# B&R Automation Studio project PrintMarkCC_LW3
Automation Studio 4.12.4.107 SP; technology packages: Acp10Arnc0 5.23.1, mapp 5.23.1, mappView 5.23.0

## Configuration Config1

### Task classes (Cpu.sw)
```
Cyclic#4:
  Cutter <- Cutter.Cutter.prg
  ConvCtrl <- ConvCtrl.ConvCtrl.prg
  AlarmsX <- Alarms.AlarmsX.prg
DataObjects: Acp10sys
NcDataObjects: gAxMsa <- Axis.gAxMaster.gAxMsa.dob, gAxMsi <- Axis.gAxMaster.gAxMsi.dob, acp10etxen <- Axis.acp10etxen.dob, gAxSlavea <- Axis.gAxSlave.gAxSlavea.dob, gAxSlavei <- Axis.gAxSlave.gAxSlavei.dob
Binaries: arsvcreg, udbdef, TCData, FWRules, Acp10map, acp10cfg, ashwd, slaveaxis, ashwac, User, sysconf, asfw, arconfig, masteraxis, iomap, Role
Libraries: Acp10man, Acp10par, NcGlobal, MpAxis, Acp10_MC, MpBase, MpCom, sys_lib, brsystem, runtime, MC_RegMa, MpAlarmX, astime, asieccon, powerlnk, asbrstr, fileio, dataobj
```

### masteraxis.mpaxisbasic - X20CP0484/Motion/masteraxis.mpaxisbasic
```
Element gmlMaster (Type=mpaxisbasic)
```

### slaveaxis.mpaxisbasic - X20CP0484/Motion/slaveaxis.mpaxisbasic
```
Element gAxisSlave (Type=mpaxisbasic)
```

## Configuration Config2

### Task classes (Cpu.sw)
```
Cyclic#1:
  Cutter <- Cutter.Cutter.prg  // cutter axis control
  ConvCtrl <- ConvCtrl.ConvCtrl.prg  // conveyor control
  AutoCtrl <- AutoCtrl.AutoCtrl.prg  // main control
Cyclic#8:
  AlarmsX <- Alarms.AlarmsX.prg  // alarm funcitons
  DataRec <- Datarec.DataRec.prg  // data recorder
DataObjects: Acp10sys
NcDataObjects: gAxMsa <- Axis.gAxMaster.gAxMsa.dob, gAxMsi <- Axis.gAxMaster.gAxMsi.dob, acp10etxen <- Axis.acp10etxen.dob, gAxSlavea <- Axis.gAxSlave.gAxSlavea.dob, gAxSlavei <- Axis.gAxSlave.gAxSlavei.dob
Binaries: arsvcreg, udbdef, TCData, FWRules, mvLoader, arflatprv, TCLang, arcoal, Acp10map, acp10cfg, ashwd, slaveaxis, ashwac, User, sysconf, asfw, arconfig, masteraxis, iomap, Role, Alarms, UserX, TC, dataReco
Libraries: Acp10man, Acp10par, NcGlobal, MpAxis, Acp10_MC, MpBase, MpCom, sys_lib, brsystem, runtime, MC_RegMa, MpAlarmX, astime, MpUserX, MpData, FileIO, DataObj, asieccon, powerlnk, asbrstr, arcert, aseth, ashw, aruser, arssl
```

### slaveaxis.mpaxisbasic - X20CP0484/Motion/slaveaxis.mpaxisbasic
```
Element gmlSlave (Type=mpaxisbasic)
```

### Alarms.mpalarmxcore - X20CP0484/mappServices/Alarms.mpalarmxcore
```
Element gAlarmXCore (Type=mpalarmxcore)
  mapp.AlarmX.Core.Configuration:
    [0]:
      Name = InTheCuttingZone
      Message = axis is inside the cutting zone please move it manually
      Code = 55
      Severity = 100
      Behavior = PersistentAlarm
    [1]:
      Name = ErrorCutting
      Code = 65
      Severity = 100
      Behavior = PersistentAlarm
```

### UserX.mpuserx - X20CP0484/mappServices/UserX.mpuserx
```
Element UserMgmtX (Type=mpuserx)
  ServerSettings:
    Server:
      AdditionalUserData:
        [0] = mail
        [1] = telephoneNumber
  Users:
    DefUser#1:
      id = admin
      name = admin
      lang = en
  Groups:
    DefGroup#1:
      id = Administrators
      level = 100
      admin = TRUE
      rights:
        [0] = FullAccess
    DefGroup#2:
      id = Everyone
    DefGroup#3:
      id = Operator
      level = 80
      rights:
        [0] = FullAccess
    DefGroup#4:
      id = Service
      level = 50
      rights:
        [0] = FullAccess
```

## Configuration Config3

### Task classes (Cpu.sw)
```
Cyclic#1:
  Cutter <- Cutter.Cutter.prg  // cutter axis control
  ConvCtrl <- ConvCtrl.ConvCtrl.prg  // conveyor control
  AutoCtrl <- AutoCtrl.AutoCtrl.prg  // main control
Cyclic#8:
  AlarmsX <- Alarms.AlarmsX.prg  // alarm funcitons
  DataRec <- Datarec.DataRec.prg  // data recorder
DataObjects: Acp10sys
NcDataObjects: gAxMsa <- Axis.gAxMaster.gAxMsa.dob, gAxMsi <- Axis.gAxMaster.gAxMsi.dob, acp10etxen <- Axis.acp10etxen.dob, gAxSlavea <- Axis.gAxSlave.gAxSlavea.dob, gAxSlavei <- Axis.gAxSlave.gAxSlavei.dob
Binaries: arsvcreg, udbdef, TCData, FWRules, mvLoader, arflatprv, TCLang, arcoal, Acp10map, acp10cfg, ashwd, slaveaxis, ashwac, User, sysconf, asfw, arconfig, masteraxis, iomap, Role, Alarms, UserX, TC, dataReco
Libraries: Acp10man, Acp10par, NcGlobal, MpAxis, Acp10_MC, MpBase, MpCom, sys_lib, brsystem, runtime, MC_RegMa, MpAlarmX, astime, MpUserX, MpData, FileIO, DataObj, asieccon, powerlnk, arcert, aseth, ashw, aruser, arssl, AsBrStr, MpServer, MpPackML
```

### Acp10map.ncm - X20CP0484/Motion/Acp10map.ncm
```
NcMapping (NcSwId=Acp10, DisabledNodesAreHidden=False)
  NcObject gAxSlave (ModuleId=8V1010.00-2a, Type=ncAXIS, Channel=1, AcoposSimulation=Off, InitParameter=gAxSlavei, AcoposParameter=gAxSlavea, AdditionalData=PLCopen_ModPos="3600,1" , Disabled=FALSE, ModuleDisabled=FALSE)
  NcObject 8V1010.00-2a_ncV_AXIS1 (ModuleId=8V1010.00-2a, Type=ncV_AXIS, Channel=1, Disabled=TRUE, ModuleDisabled=FALSE)
  NcObject gAxMaster (ModuleId=8V1010.00-2, Type=ncAXIS, Channel=1, AcoposSimulation=Off, InitParameter=gAxMsi, AcoposParameter=gAxMsa, Disabled=FALSE, ModuleDisabled=FALSE)
  NcObject 8V1010.00-2_ncV_AXIS1 (ModuleId=8V1010.00-2, Type=ncV_AXIS, Channel=1, Disabled=TRUE, ModuleDisabled=FALSE)
```

### slaveaxis.mpaxisbasic - X20CP0484/Motion/slaveaxis.mpaxisbasic
```
Element gmlSlave (Type=mpaxisbasic)
  Alarms = MpAlarmX
```

### UserX.mpuserx - X20CP0484/mappServices/UserX.mpuserx
```
Element UserMgmtX (Type=mpuserx)
  ServerSettings:
    Server:
      AdditionalUserData:
        [0] = mail
        [1] = telephoneNumber
  Users:
    DefUser#1:
      id = admin
      name = admin
      lang = en
    DefUser#2:
      id = operator
      name = operator
      lang = en
  Groups:
    DefGroup#1:
      id = Administrators
      level = 100
      admin = TRUE
      rights:
        [0] = FullAccess
    DefGroup#2:
      id = Everyone
    DefGroup#3:
      id = Operator
      level = 80
      rights:
        [0] = FullAccess
    DefGroup#4:
      id = Service
      level = 50
      rights:
        [0] = FullAccess
```

### mlPack.mppackmlcore - X20CP0484/mappServices/mlPack.mppackmlcore
```
Element gPackMLCore (Type=mppackmlcore)
  Modes:
    Mode[1]:
      ModeID = 1
      Name = Production
```

## Logical view

Binary libraries used (declarations not repeated): operator, runtime, astime, AsIecCon, Acp10man, Acp10par, NcGlobal, MpAxis, Acp10_MC, MpBase, MpCom, sys_lib, brsystem, MC_RegMa, MpAlarmX, MpUserX, MpData, FileIO, DataObj

### Global.typ - Global data types
```iecst
(*main control*)

TYPE
	AxisCtrl_typ : 	STRUCT  (*Axis Ctrl Struture*)
		Cmd : AxisCmd_typ; (*Axis Ctrl CMd type*)
		Para : AxisPara_typ; (*Axis para type*)
		Status : AxisStatus_typ; (*Axis Status Type*)
	END_STRUCT;
END_TYPE

(*commands*)

TYPE
	AxisCmd_typ : 	STRUCT  (*Axis Ctrl CMd type*)
		Start : BOOL; (*Start Cmd*)
		Stop : BOOL; (*Stop cmd*)
		PrintMark : BOOL; (*Print mark detection bit*)
		ErrorReset : BOOL; (*Error reset*)
		AutoMode : BOOL; (*AutoMode*)
		JogFwd : BOOL; (*Jog forward command*)
		JogBack : BOOL; (*jog BAckward c0mmand*)
		Home : BOOL; (*home Cmd*)
		SingleCutter : BOOL;
	END_STRUCT;
END_TYPE

(*parameters*)

TYPE
	AxisPara_typ : 	STRUCT  (*Axis para type*)
		Speed : UINT; (*Axis Speed*)
	END_STRUCT;
END_TYPE

(*status*)

TYPE
	AxisStatus_typ : 	STRUCT  (*Axis Status*)
		JogNegReady : BOOL; (*Axis jog neg ready status*)
		JogPosReady : BOOL; (*axis jog pos ready Statsus*)
	END_STRUCT;
END_TYPE
```

### Global.var - Global variables
```iecst
(*Axis Variables*)
VAR
	gAxMaster : ACP10AXIS_typ; (*Master Axis*)
	gAxSlave : ACP10AXIS_typ; (*Slave Axis*) (*	gAx_Slave : AxisBasic_type; (*Slave Axis Structure*) (*gAx_Master : AxisBasic_type; MAster axis Structure*)
END_VAR
(*Automatic mode*)
VAR
	gAutoMode : BOOL; (*automatic mode for machine*)
	gManulMode : BOOL; (*manual mode for machine*)
END_VAR
(*IR trigger for conveyor belt*)
VAR
	gIR_Trigger : BOOL; (*trigger of IR for Conveyor axis master*)
END_VAR
(*for mappview commands given'*)
VAR
	gMi_ModeConfirm : BOOL; (*mode confirmation for hmi*)
	gMI_MODE : BOOL;
END_VAR
```


### Package Logical/Axis - Axis Package


- Data object Logical/Axis/gAxMaster/gAxMsa (Apt) - Conv Axis SPT (no source held here)

- Data object Logical/Axis/gAxMaster/gAxMsi (Ax) - COnv Axis Parameter Table (no source held here)

### Package Logical/Axis/gAxSlave - Cutter Axis Package

### Data object Logical/Axis/gAxSlave/gAxSlavei (Ax) - Cutter Axis Paramter table

#### gAxisSlave.ax
```
InitParameter (Version=5.23.1, NcSwId=ACP10)
  ACP10AXIS_typ:
    dig_in:
      level:
        reference = ncACTIV_HI
        pos_hw_end = ncACTIV_HI
        neg_hw_end = ncACTIV_HI
        trigger1 = ncACTIV_HI
        trigger2 = ncACTIV_HI
    encoder_if:
      parameter:
        count_dir = ncSTANDARD
        scaling:
          load:
            units = 3600
            rev_motor = 1
    limit:
      parameter:
        v_pos = 108000.0
        v_neg = 108000.0
        a1_pos = 1080000.0
        a2_pos = 1080000.0
        a1_neg = 1080000.0
        a2_neg = 1080000.0
        t_jolt = 0.18
        t_in_pos = 0.0
        pos_sw_end = 8388607
        neg_sw_end = -8388608
        ds_warning = 180.0
        ds_stop = 360.0
        a_stop = 1.0E+30
        dv_stop = 0.0
        dv_stop_mode = ncOFF
    controller:
      mode = ncPOSITION + ncFF
      position:
        kv = 295.0
        tn = 0.0
        t_predict = 0.0004
        t_total = 0.0004
        p_max = 1.0E+30
        i_max = 0.0
      speed:
        kv = 0.6
        tn = 0.0
        t_filter = 0.0
        isq_filter1:
          type = ncOFF
          a0 = 0.0
          a1 = 0.0
          b0 = 0.0
          b1 = 0.0
          b2 = 0.0
          c0_par_id = 0
          c1_par_id = 0
        isq_filter2:
          type = ncOFF
          a0 = 0.0
          a1 = 0.0
          b0 = 0.0
          b1 = 0.0
          b2 = 0.0
          c0_par_id = 0
          c1_par_id = 0
        isq_filter3:
          type = ncOFF
          a0 = 0.0
          a1 = 0.0
          b0 = 0.0
          b1 = 0.0
          b2 = 0.0
          c0_par_id = 0
          c1_par_id = 0
      uf:
        type = ncLINEAR + ncCORRECTION
        auto_config = ncMOTOR_PAR
        u0 = 0.0
        un = 0.0
        fn = 50.0
        k_f_slip = 0.0
      ff:
        mode = ncSTANDARD
        torque_load = 0.0
        torque_pos = 0.00623549
        torque_neg = 0.00399368
        kv_torque = 0.0016169
        inertia = 9.44476E-05
        t_filter_a = 0.0
      fb:
        mode = ncSTANDARD
        speed_mix_ratio = 0.0
        speed_kv = 0.0
      model:
        mass1:
          inertia = 0.0
          viscous_friction = 0.0
        mass2:
          inertia = 0.0
          viscous_friction = 0.0
          stiffness = 0.0
          damping = 0.0
    move:
      stop:
        parameter[0]:
          decel_ramp = ncA_LIMIT
          controller = ncON
        parameter[1]:
          decel_ramp = ncA_LIMIT
          controller = ncON
        parameter[2]:
          decel_ramp = ncA_LIMIT
          controller = ncON
        parameter[3]:
          decel_ramp = ncA_LIMIT
          controller = ncON
        quickstop:
          decel_ramp = ncA_LIMIT
          t_jolt = 0.0
        drive_error:
          decel_ramp = ncA_LIMIT
      homing:
        parameter:
          s = 0
          v_switch = 5000.0
          v_trigger = 500.0
          a = 50000.0
          mode = ncDIRECT
          edge_sw = ncPOSITIVE
          start_dir = ncPOSITIVE
          trigg_dir = ncPOSITIVE
          ref_pulse = ncOFF
          fix_dir = ncOFF
          tr_s_block = 0.0
          torque_lim = 0.0
          ds_block = 0.0
          ds_stop = 0.0
      basis:
        parameter:
          v_pos = 500.0
          v_neg = 5000.0
          a1_pos = 50000.0
          a2_pos = 50000.0
          a1_neg = 50000.0
          a2_neg = 50000.0
    message:
      text:
        parameter:
          format = ncBREAK + ncZERO
          columns = 80
          data_modul = acp10etxen
```

### Program Logical/Cutter/Cutter (IEC)

#### Main.st - Init, cyclic, exit code
```iecst
(*|ŻŻŻŻŻŻŻŻŻŻŻŻŻŻŻŻŻŻŻŻŻŻŻŻŻŻŻŻŻŻŻŻŻŻŻŻŻŻŻŻŻŻŻŻŻŻŻŻŻŻŻŻŻŻŻŻŻŻŻŻŻŻŻŻŻŻŻŻŻŻŻŻŻŻŻŻŻŻŻŻŻŻŻŻŻŻŻŻŻŻŻŻŻŻŻŻŻŻŻŻŻŻŻŻŻŻŻŻŻŻ|*)
(*| Copyright      :-  B&R Industrial Automation GmbH															 |*)
(*| Contact Person :-  maskeu																					 |*)
(*|——————————————————————————————————————————————————————————————————————————————————————————————————————————————|*)
(*| System       :-  cutter control                                                                    	 		 |*)
(*| Task Name    :-  cutter control																		  		 |*)
(*| Auther Name  :-  maskeu																						 |*)
(*| Created Date :-  December 19, 2023 																		   	 |*)
(*| Task Class   :-  Task Class# 1                                                                 				 |*)
(*| Task Time    :-  Task Timing 2mSec                                                                           |*)
(*| OS Version   :-  G4.93                                                                                       |*)
(*| AS Version   :-  AS 4.12.4.107 SP                                                                            |*)
(*|——————————————————————————————————————————————————————————————————————————————————————————————————————————————|*)
(*| Description  :-  CUTTER cam sequnce and basic initial prameters		    									 |*)
(*| V1.00.0   19/12/2023	 Maskeu        added cam sequnce 									Complete		 |*)
(*| V2.00.0   21/12/2023	 Maskeu        added basic parameters for axis						Complete		 |*)
(*| V3.00.0   22/12/2023	 Maskeu        added reg capture parameters 						Complete		 |*)
PROGRAM _INIT

	//providing initial parameters
	iBasicParSlave.Acceleration:=10800;
	iBasicParSlave.Deceleration:=108000;
	iBasicParSlave.Jog.Deceleration:=108000;
	iBasicParSlave.Jog.Acceleration:=108000;
	iBasicParSlave.Jog.Velocity:=360;

	//assigning reg capture prameters
	iRegCapAdvPar.EventSourceParID := ACP10PAR_STAT_TRIGGER1;
	iRegCapAdvPar.Edge := ncP_EDGE;
	iRegCapAdvPar.MinWidth := 50;
	iRegCapAdvPar.MaxWidth := 200;
	iRegCapAdvPar.WindowNeg := 200;
	iRegCapAdvPar.WindowPos := 200;
	iRegCapAdvPar.SensorDelay := 200;
	iRegCapAdvPar.CorrectCurrentCycle := TRUE;
	iRegCapAdvPar.CorrectionValueLimitNeg := 70;
	iRegCapAdvPar.CorrectionValueLimitPos := 70;

	iRegCapConfig.DistanceToSensor := 1050; //distance betwwen ir sensor to cutter
	iRegCapConfig.ProductLength := 700;		//length of the product
	iRegCapConfig.RegMarkPosition := 700;	//reg par at positon 7c,
	iRegCapConfig.RegMarkOffset := 10;		//offset value
END_PROGRAM

PROGRAM _CYCLIC
	IF iCutCtrl.Cmd.SingleCutter THEN
		//axis control  in single mode
		SingleCutter;
		// cam for single cutter
		CamSingle;
	ELSE
		//axis control  in dual mode
		MultCutter;
		// cam for Dual Cutter
		CamMulti;
	END_IF

	IF iFb_SlaveAx.Info.PLCopenState = mpAXIS_SYNCHRONIZED_MOTION THEN
		iFb_RegCap();
	END_IF

	//reg capturing action
	RegCap;

	//linking the slave to cam sequence
	iFb_CamSequ.MpLink :=ADR(gmlSlave);
	iFb_CamSequ.Enable :=TRUE;

	//parameters for cam seqeunce
	iFb_CamSequ.Parameters :=ADR(iAx_CamSequence);

	//linking the master with cam sequence
	iFb_CamSequ.MpLinkMaster :=ADR(gmlMaster);
	iFb_CamSequ.StartSequence :=iFb_CamSequ.Info.MasterReady AND iFb_CamSequ.Info.SlaveReady;

	//fucniton block is callled
	iFb_CamSequ();

	IF (iMI_CutSetJogAcc <> (iBasicParSlave.Jog.Acceleration * PER_SEC)/PRODUCT_LENGTH
		OR iMI_CutSetJogDeacc <> (iBasicParSlave.Jog.Deceleration  * PER_SEC)/PRODUCT_LENGTH
		OR iMI_CutSetJogVel <> (iBasicParSlave.Jog.Velocity * PER_SEC)/PRODUCT_LENGTH)
		AND NOT gMI_MODE THEN
		iFb_SlaveAx.Update := TRUE;
		IF iFb_SlaveAx.UpdateDone THEN
			iFb_SlaveAx.Update := FALSE;
		END_IF
	END_IF

	iBasicParSlave.Jog.Acceleration := (iMI_CutSetJogAcc * PRODUCT_LENGTH)/PER_SEC;
	iBasicParSlave.Jog.Deceleration := (iMI_CutSetJogDeacc * PRODUCT_LENGTH)/PER_SEC;
	iBasicParSlave.Jog.Velocity := (iMI_CutSetJogVel * PRODUCT_LENGTH)/PER_SEC;

	iMI_CutActSpeed := (iFb_SlaveAx.Velocity * PER_SEC)/PRODUCT_LENGTH ;
END_PROGRAM

PROGRAM _EXIT

	//disabling all the functions
	iFb_AxisSlave.Enable:=FALSE;
	iFb_AxisSlave();
	iFb_CamSequ.Enable:=FALSE;
	iFb_CamSequ();
END_PROGRAM
```

#### Types.typ - Local data types
```iecst
(*jog limiting enumeration*)

TYPE
	Joglim_enum :
		( (*jog limit state enumeration*)
		enCHECKVEL, (*Checking value*)
		enADDVEL, (*gicing jog values*)
		enUPPERPOS, (*upper position state*)
		enLOWERPOS, (*lower position state*)
		enUPDATE, (*updating the state according position*)
		enRESET (*reseting the values*)
		);
END_TYPE

(*axis steps enumeration*)

TYPE
	AxStep_enum :
		( (*axis enumeration*)
		enINITA, (*initiate*)
		enSTARTA, (*starting axis*)
		enNEEGHOMEMOVE, (*negative direction homing*)
		enPOWER_ONA, (*powering on*)
		enPOSHOMINGSEC, (*positive direction homing*)
		enPOSHOMING, (*positive side homing*)
		enNEGHOMING, (*negative side homing*)
		enHOMEA, (*homing state*)
		enOPERATIONA, (*operation state*)
		enERRORA, (*error state*)
		enMANUAL, (*manual mode is on*)
		enAUTOMATIC, (*automatic mode is on*)
		enJOGPOSITIVE, (*jog positive state*)
		enJOGNEGATIVE, (*jog backward state*)
		enCUTTINGZONE (*cutting zone*)
		);
END_TYPE
```

#### Variables.var - Local variables
```iecst
VAR
	iVl_OldAcc : REAL; (*old accelartion *)
	iMi_LogoNegDir : BOOL; (*negtive direction hmi button*)
	icmdUpdate : BOOL; (*update command*)
	icmdPower : BOOL; (*powering on the axis*)
	icmdHome : BOOL; (*hooming the axis*)
END_VAR
VAR RETAIN
	icmdMoveVelocity : BOOL; (*move velocity for axis*)
END_VAR
VAR
	icmdMoveAdditive : BOOL; (*move additive axis*)
END_VAR
VAR RETAIN
	icmdStop : BOOL; (*stopping the axis*)
END_VAR
VAR
	iVl_OldAccNeg : REAL; (*old accelation for axis*)
	icmdErrorReset : BOOL; (*error reseting the axis*)
	iVl_OldVelocity : REAL; (*old velocity for logo  conveyor*)
END_VAR
(*all the strucutres*)
VAR
	iFb_MC_MoveVelocity_0 : MC_MoveVelocity; (*funciton bloack for velocity*)
	iFb_SlaveAx : MpAxisBasic; (*basic function for axis*)
	iBasicParSlave : MpAxisBasicParType; (*basic parameters for axis*)
	iParaSlave : MpAxisBasicParType; (*paraemeters for slave*)
	iCutCtrl : AxisCtrl_typ; (*cutter control*)
	iParamMaster : MpAxisBasicParType; (*parameters for master*)
	iAx_CamSequence : MpAxisCamSequencerParType; (*Cam Seq Structure*)
	iJogLimState : Joglim_enum; (*jog limit enumeration*)
	iAxStep_enum : AxStep_enum; (*steps for logo conveyor*)
END_VAR
(*All the funciton blocks*)
VAR
	iFb_AxisSlave : MpAxisBasic; (*fucniton block for axis slave*)
	iFb_AxisMater : MpAxisBasic; (*fucniton block for axis master*)
	iFb_CamSequ : MpAxisCamSequencer; (*cam sequencer fucniton block*)
	iFb_RegCap : MC_BR_RegMarkCapture002; (*reg capture funciton*)
	iRegCapAdvPar : MC_BR_ADV_RM2_REF; (*reg capture parameters*)
	iRegCapConfig : MC_BR_CFG_RM2_REF; (*reg capture configuration*)
	iAbsVal : LREAL; (*absolute value for homing downside*)
	icmdMoveAbsoulte : BOOL; (*move absoulte commands*)
END_VAR
(*Al the constatnt for homing , position , offset value etc.*)
VAR CONSTANT
	HOMING_VEL : REAL := 500; (*homing velocity*)
	HOFFSET_SINGLE : REAL := 1033; (*offset for single cutter*)
	SPEED : REAL := 0.25; (*speed*)
	ZEROSPD : REAL := 0; (*zero speed to assign*)
	SCALSPEEDTEN : REAL := 10000; (*scaling of speed*)
	START_VEL : REAL := 145;
	INIT_FIHNRD : REAL := 500; (*inital value five hundread*)
	INIT_FTHOUSAND : REAL := 5000; (*inital five thousand *)
	INIT_THOUSAND : REAL := 1000; (*inital value thousand*)
	UPPER_CUT_POS : REAL := 3013; (*upper cutting position for first cutter*)
END_VAR
VAR
	HOFFSET_DUAL : REAL := 133; (*offset value for homing*)
END_VAR
VAR CONSTANT
	LOWER_CUT_POS : REAL := 2653; (*lower cutting position for second cutter*)
	HOFFSET_NEGDUAL : LREAL := 33; (*offset for negative ohming in dual cutter*)
	FIRST_CUT_UPPER : LREAL := 3013; (*first cutter upper positon of cutting*)
	HOME_POS : LREAL := 1933; (*homing positon downside*)
	SEC_CUT_UPPER : LREAL := 1213; (*second cutter upper cut position*)
	FIRST_CUT_LOWER : LREAL := 2653; (*first cutter lower positon*)
	MAX_POS_AXIS : LREAL := 3599; (*max axis positon*)
	SEC_CUT_LOWER : LREAL := 853; (*second cutter lower value*)
	HOME_OFFSET : LREAL := 133; (*offset value for homing*)
END_VAR
VAR
	LOWER_BUFER : LREAL := 0; (*lower buffer value*)
	ZERO : LREAL := 0; (*zero vlaue*)
END_VAR
VAR CONSTANT
	PRODUCT_LENGTH : REAL := 700.0; (*Product length*)
	PER_SEC : REAL := 60.0; (*Per Sec*)
END_VAR
(*HMI varible*)
VAR
	iMI_CutSetJogAcc : REAL := 300; (*Cut set jog acceleration*)
	iMI_CutSetJogDeacc : REAL := 300; (*Cut jog deacceleration*)
	iMI_CutActSpeed : REAL; (*Cut act speed*)
	iMI_CutSetJogVel : REAL := 45; (*Cut set jog velocity*)
END_VAR
```

#### SingCutter.st - single cutter control
```iecst
(*|ŻŻŻŻŻŻŻŻŻŻŻŻŻŻŻŻŻŻŻŻŻŻŻŻŻŻŻŻŻŻŻŻŻŻŻŻŻŻŻŻŻŻŻŻŻŻŻŻŻŻŻŻŻŻŻŻŻŻŻŻŻŻŻŻŻŻŻŻŻŻŻŻŻŻŻŻŻŻŻŻŻŻŻŻŻŻŻŻŻŻŻŻŻŻŻŻŻŻŻŻŻŻŻŻŻŻŻŻŻŻ|*)
(*| Copyright      :-  B&R Industrial Automation GmbH															 |*)
(*| Contact Person :-  maskeu																					 |*)
(*|——————————————————————————————————————————————————————————————————————————————————————————————————————————————|*)
(*| System       :-  cutter control                                                                    	 		 |*)
(*| Task Name    :-  cutter control																		  		 |*)
(*| Auther Name  :-  maskeu																						 |*)
(*| Created Date :-  December 19, 2023 																		   	 |*)
(*| Task Class   :-  Task Class# 1                                                                 				 |*)
(*| Task Time    :-  Task Timing 2mSec                                                                           |*)
(*| OS Version   :-  G4.93                                                                                       |*)
(*| AS Version   :-  AS 4.12.4.107 SP                                                                            |*)
(*|——————————————————————————————————————————————————————————————————————————————————————————————————————————————|*)
(*| Description  :-  CUTTER cam sequnce and basic initial prameters		    									 |*)
(*| V1.00.0   19/12/2023	 Maskeu        added homing states									Complete		 |*)
(*| V2.00.0   20/12/2023	 Maskeu        added jog limits										Complete		 |*)
(*| V3.00.0   23/12/2023	 Maskeu        modified positive homing state						Complete		 |*)

ACTION SingleCutter:
	//linking the motor with axis
	gIR_Trigger:=iFb_SlaveAx.Info.DigitalInputsStatus.Trigger1;
	iFb_SlaveAx.Enable := 1;
	iFb_SlaveAx.MpLink := ADR(gmlSlave);
	iFb_SlaveAx.Axis := ADR(gAxSlave);

	iFb_SlaveAx.Parameters := ADR(iBasicParSlave);
	iFb_SlaveAx();

	//	if new velocity by user input is different then will update
	//	IF iVl_OldVelocity <> iBasicParSlave.Acceleration THEN
	//		iFb_SlaveAx.Update:=TRUE ;
	//		IF	iFb_SlaveAx.UpdateDone=TRUE THEN
	//			iVl_OldVelocity:= iBasicParSlave.Velocity;
	//			iFb_SlaveAx.Update:=FALSE ;
	//		END_IF;
	//	END_IF;
	//
	//	//	if new accelaration by user input is different then will update
	//	IF iVl_OldAcc<> iBasicParSlave.Acceleration THEN
	//		iFb_SlaveAx.Update:=TRUE ;
	//		IF	iFb_SlaveAx.UpdateDone=TRUE THEN
	//			iVl_OldAcc:= iBasicParSlave.Acceleration;
	//			iFb_SlaveAx.Update:=FALSE ;
	//		END_IF;
	//	END_IF;
	//
	//	//	if new deccelaration by user input is different then will update
	//	IF iVl_OldAccNeg<> iBasicParSlave.Deceleration THEN
	//		iFb_SlaveAx.Update:=TRUE ;
	//		IF	iFb_SlaveAx.UpdateDone=TRUE THEN
	//			iVl_OldAccNeg:= iBasicParSlave.Deceleration;
	//			iFb_SlaveAx.Update:=FALSE ;
	//		END_IF;
	//	END_IF;

	//Limit for the torque
	iBasicParSlave.Torque.Limit:=0.8;

	//stopping the axis command
	IF icmdStop=TRUE THEN
		iFb_SlaveAx.Stop:=TRUE;
		IF iFb_SlaveAx.Stopped=TRUE THEN
			iFb_SlaveAx.Stop:=FALSE;
			icmdStop:=FALSE;
		END_IF;
	END_IF;

	//if axis is in error mode
	IF iFb_SlaveAx.Error=TRUE THEN
		iAxStep_enum:=enERRORA;
	END_IF;

	//state neumeration for axis
	CASE iAxStep_enum OF

		//initializtion
		enINITA:
			IF iCutCtrl.Cmd.Start=TRUE THEN
				iAxStep_enum := 	enSTARTA;
			END_IF;
			//starting
		enSTARTA:
			IF iFb_SlaveAx.Info.ReadyToPowerOn = TRUE THEN
				iAxStep_enum := enPOWER_ONA;
			END_IF

			//poweron the axis
		enPOWER_ONA:
			iFb_SlaveAx.Power := TRUE;
			IF iFb_SlaveAx.PowerOn = TRUE THEN

				//when axis has passed lower cut positon
				IF iFb_SlaveAx.PowerOn AND iFb_SlaveAx.Position < LOWER_CUT_POS THEN
					iFb_SlaveAx.Update:=TRUE;
					IF iFb_SlaveAx.UpdateDone=TRUE THEN
						iAxStep_enum := enNEGHOMING;
						iFb_SlaveAx.Update:=FALSE;
					END_IF;
				END_IF

				//when axis has not passed upper cut positon
				IF iFb_SlaveAx.PowerOn AND iFb_SlaveAx.Position > UPPER_CUT_POS THEN
					iFb_SlaveAx.Update:=TRUE;
					IF iFb_SlaveAx.UpdateDone=TRUE THEN
						iAxStep_enum := enPOSHOMING;
						iFb_SlaveAx.Update:=FALSE;
					END_IF;
				END_IF
			END_IF

			//homing in positive direction
		enNEGHOMING:
			iBasicParSlave.Home.Mode:=mpAXIS_HOME_MODE_REF_PULSE;
			iBasicParSlave.Home.HomingDirection:=mpAXIS_HOME_DIR_NEGATIVE;
			iBasicParSlave.Home.SensorOffset := HOFFSET_SINGLE;
			iBasicParSlave.Home.HomingVelocity := HOMING_VEL;
			iBasicParSlave.Home.StartVelocity := START_VEL;
			iFb_SlaveAx.Home := TRUE;
			iAxStep_enum:=	enOPERATIONA;

			//homing in negative direction
		enPOSHOMING:
			iBasicParSlave.Home.Mode:=mpAXIS_HOME_MODE_REF_PULSE;
			iBasicParSlave.Home.HomingDirection:=mpAXIS_HOME_DIR_POSITIVE;;
			iBasicParSlave.Home.SensorOffset := HOFFSET_SINGLE;
			iBasicParSlave.Home.HomingVelocity := HOMING_VEL;
			iBasicParSlave.Home.StartVelocity := START_VEL;
			iFb_SlaveAx.Home := TRUE;
			iAxStep_enum:=	enOPERATIONA;
			//operation mode
		enOPERATIONA:

			IF iFb_SlaveAx.IsHomed=TRUE THEN
				iFb_SlaveAx.Home := FALSE;
				iAxStep_enum:=enOPERATIONA;
				IF gAutoMode=TRUE THEN

				ELSIF gManulMode THEN
					iAxStep_enum:=	enMANUAL;
				END_IF;
			END_IF;

		enMANUAL:
			IF iCutCtrl.Cmd.JogFwd THEN
				iAxStep_enum:=	enJOGPOSITIVE;
			END_IF;
			IF iCutCtrl.Cmd.JogBack THEN
				iAxStep_enum:=	enJOGNEGATIVE;
			END_IF;

			IF iFb_SlaveAx.Position = FIRST_CUT_LOWER THEN
				iCutCtrl.Cmd.JogFwd := FALSE;
			END_IF
		enJOGPOSITIVE:
			IF NOT iCutCtrl.Cmd.JogFwd=TRUE OR iFb_SlaveAx.Position=FIRST_CUT_LOWER THEN
				iFb_SlaveAx.JogPositive:=FALSE;
				iAxStep_enum:=enOPERATIONA;
			ELSE
				iFb_SlaveAx.JogPositive:=TRUE;
			END_IF;

			IF iFb_SlaveAx.Position= FIRST_CUT_LOWER THEN
				iCutCtrl.Cmd.JogFwd:=FALSE;
			END_IF;

		enJOGNEGATIVE:
			IF NOT iCutCtrl.Cmd.JogBack=TRUE OR iFb_SlaveAx.Position=FIRST_CUT_UPPER THEN
				iFb_SlaveAx.JogNegative:=FALSE;
				iAxStep_enum:=enOPERATIONA;
			ELSE
				iFb_SlaveAx.JogNegative:=TRUE;
			END_IF;

			IF iFb_SlaveAx.Position= FIRST_CUT_UPPER THEN
				iCutCtrl.Cmd.JogBack:=FALSE;
			END_IF;

		enCUTTINGZONE:
			iFb_SlaveAx.Power:=FALSE;
			IF (iFb_SlaveAx.Position < FIRST_CUT_LOWER OR iFb_SlaveAx.Position  >FIRST_CUT_UPPER) AND iFb_SlaveAx.IsHomed THEN
				iFb_SlaveAx.Power:=TRUE;
				iAxStep_enum := enOPERATIONA;
			ELSIF  (iFb_SlaveAx.Position  < FIRST_CUT_LOWER OR iFb_SlaveAx.Position  >FIRST_CUT_UPPER) AND NOT  iFb_SlaveAx.IsHomed THEN
				iAxStep_enum := enPOWER_ONA;
			END_IF
			//error mode
		enERRORA:
			iFb_SlaveAx.Power := FALSE;
			icmdMoveVelocity := FALSE;
			icmdStop := FALSE;

			icmdErrorReset:=TRUE;
			IF iFb_SlaveAx.Error = FALSE THEN;
				iAxStep_enum := enSTARTA;
				icmdErrorReset := FALSE;
			END_IF
	END_CASE

	CASE iJogLimState OF

		//checking the value of jog positive and negative
		enCHECKVEL:
			IF iFb_SlaveAx.JogNegative = TRUE THEN
				iJogLimState							:= enUPPERPOS;
			END_IF;
			IF (iFb_SlaveAx.JogPositive = TRUE) THEN
				iJogLimState							:= enLOWERPOS;
			END_IF;

			//will give command once again
		enADDVEL:
			iFb_SlaveAx.JogPositive						:= TRUE;
			iFb_SlaveAx.JogNegative						:= TRUE;
			iJogLimState								:= enCHECKVEL;

			//if axis position is greater than upper cut
		enUPPERPOS:
			IF (iFb_SlaveAx.CommandAborted = TRUE) THEN
				iJogLimState							:= enADDVEL;
				iFb_SlaveAx.JogNegative	:= FALSE;
			END_IF;

			IF (iFb_SlaveAx.Position > UPPER_CUT_POS)THEN
				iBasicParSlave.Jog.LowerLimit			:= FIRST_CUT_UPPER;
				iBasicParSlave.Jog.UpperLimit			:= MAX_POS_AXIS;
				iFb_SlaveAx.Update						:= TRUE;
				iJogLimState							:= enUPDATE;
			END_IF;

			//if axis position is lower than lower cut
		enLOWERPOS:
			IF (iFb_SlaveAx.CommandAborted = TRUE) THEN
				iJogLimState							:= enADDVEL;
				iFb_SlaveAx.JogPositive					:= FALSE;
			END_IF;

			IF (iFb_SlaveAx.Position < LOWER_CUT_POS)THEN
				iBasicParSlave.Jog.LowerLimit			:=ZERO;
				iBasicParSlave.Jog.UpperLimit			:= FIRST_CUT_LOWER;
				iFb_SlaveAx.Update						:= TRUE;
				iJogLimState							:= enUPDATE;
			END_IF;

			//updating state on position
		enUPDATE:
			IF iFb_SlaveAx.UpdateDone = TRUE THEN
				iFb_SlaveAx.Update						:= FALSE;
			END_IF;
			IF iFb_SlaveAx.JogNegative = TRUE AND iFb_SlaveAx.Position <ZERO AND iFb_SlaveAx.Position > UPPER_CUT_POS THEN
				iJogLimState							:= enUPPERPOS;
			END_IF;
			IF (iFb_SlaveAx.JogPositive = TRUE) AND iFb_SlaveAx.Position > ZERO AND iFb_SlaveAx.Position < LOWER_CUT_POS  THEN
				iJogLimState							:= enLOWERPOS;
			END_IF;
			IF ((iFb_SlaveAx.Position = FIRST_CUT_UPPER) OR (iFb_SlaveAx.Position =FIRST_CUT_LOWER )) THEN
				iFb_SlaveAx.JogNegative					:= FALSE;
				iFb_SlaveAx.JogPositive					:= FALSE;
				iJogLimState							:= enRESET;
			END_IF;

			//reseting the values
		enRESET:

			iBasicParSlave.Jog.LowerLimit				:= ZERO;
			iBasicParSlave.Jog.UpperLimit				:= ZERO;
			iFb_SlaveAx.Update							:= TRUE;
			IF iFb_SlaveAx.UpdateDone = TRUE THEN
				iFb_SlaveAx.Update						:= FALSE;
				iJogLimState							:= enCHECKVEL;
			END_IF;
	END_CASE;

	iBasicParSlave.CyclicRead.TorqueMode			:=mpAXIS_READ_CYCLIC;
	//Reset Condition
	IF iCutCtrl.Cmd.Start= FALSE THEN
		iAxStep_enum 			:= enINITA;
		iJogLimState 			:= enCHECKVEL;
	END_IF

END_ACTION
```

#### MultCutter.st - multi cutter control
```iecst
(*|ŻŻŻŻŻŻŻŻŻŻŻŻŻŻŻŻŻŻŻŻŻŻŻŻŻŻŻŻŻŻŻŻŻŻŻŻŻŻŻŻŻŻŻŻŻŻŻŻŻŻŻŻŻŻŻŻŻŻŻŻŻŻŻŻŻŻŻŻŻŻŻŻŻŻŻŻŻŻŻŻŻŻŻŻŻŻŻŻŻŻŻŻŻŻŻŻŻŻŻŻŻŻŻŻŻŻŻŻŻŻ|*)
(*| Copyright      :-  B&R Industrial Automation GmbH															 |*)
(*| Contact Person :-  maskeu																					 |*)
(*|——————————————————————————————————————————————————————————————————————————————————————————————————————————————|*)
(*| System       :-  cutter control                                                                    	 		 |*)
(*| Task Name    :-  cutter control																		  		 |*)
(*| Auther Name  :-  maskeu																						 |*)
(*| Created Date :-  December 19, 2023 																		   	 |*)
(*| Task Class   :-  Task Class# 1                                                                 				 |*)
(*| Task Time    :-  Task Timing 2mSec                                                                           |*)
(*| OS Version   :-  G4.93                                                                                       |*)
(*| AS Version   :-  AS 4.12.4.107 SP                                                                            |*)
(*|——————————————————————————————————————————————————————————————————————————————————————————————————————————————|*)
(*| Description  :-  Multiple cutter fucnitoning		    													 |*)
(*| V1.00.0   19/12/2023	 Maskeu        added homing states									Complete		 |*)
(*| V2.00.0   21/12/2023	 Maskeu        added homing for lower positon with absolute homing	Complete		 |*)

ACTION MultCutter:
	//linking the motor with axis
	gIR_Trigger:=iFb_SlaveAx.Info.DigitalInputsStatus.Trigger1;
	iFb_SlaveAx.Enable := 1;
	iFb_SlaveAx.MpLink := ADR(gmlSlave);
	iFb_SlaveAx.Axis := ADR(gAxSlave);

	iFb_SlaveAx.Parameters := ADR(iBasicParSlave);
	iFb_SlaveAx();

	//	if new velocity by user input is different then will update
	//	IF iVl_OldVelocity <> iBasicParSlave.Acceleration THEN
	//		iFb_SlaveAx.Update:=TRUE ;
	//		IF	iFb_SlaveAx.UpdateDone=TRUE THEN
	//			iVl_OldVelocity:= iBasicParSlave.Velocity;
	//			iFb_SlaveAx.Update:=FALSE ;
	//		END_IF;
	//	END_IF;
	//
	//	//	if new accelaration by user input is different then will update
	//	IF iVl_OldAcc<> iBasicParSlave.Acceleration THEN
	//		iFb_SlaveAx.Update:=TRUE ;
	//		IF	iFb_SlaveAx.UpdateDone=TRUE THEN
	//			iVl_OldAcc:= iBasicParSlave.Acceleration;
	//			iFb_SlaveAx.Update:=FALSE ;
	//		END_IF;
	//	END_IF;
	//
	//	//	if new deccelaration by user input is different then will update
	//	IF iVl_OldAccNeg<> iBasicParSlave.Deceleration THEN
	//		iFb_SlaveAx.Update:=TRUE ;
	//		IF	iFb_SlaveAx.UpdateDone=TRUE THEN
	//			iVl_OldAccNeg:= iBasicParSlave.Deceleration;
	//			iFb_SlaveAx.Update:=FALSE ;
	//		END_IF;
	//	END_IF;

	//Limit for the torque
	iBasicParSlave.Torque.Limit:=0.8;

	//position for the axis for homing
	iBasicParSlave.Position:=1900;

	//stopping the axis command
	IF iFb_SlaveAx.Stop=TRUE THEN
		IF iFb_SlaveAx.Stopped=TRUE THEN
			iFb_SlaveAx.Stop:=FALSE;
		END_IF;
	END_IF;

	//if axis is in error mode
	IF iFb_SlaveAx.Error=TRUE THEN
		iAxStep_enum:=enERRORA;
	END_IF;

	//state neumeration for axis
	CASE iAxStep_enum OF

		//initializtion
		enINITA:
			IF iCutCtrl.Cmd.Start=TRUE THEN
				iAxStep_enum := 	enSTARTA;
			END_IF;
			//starting
		enSTARTA:
			IF iFb_SlaveAx.Info.ReadyToPowerOn = TRUE THEN
				iAxStep_enum := enPOWER_ONA;
			END_IF

			//poweron the axis
		enPOWER_ONA:
			iFb_SlaveAx.Power := TRUE;
			IF iFb_SlaveAx.PowerOn = TRUE THEN
				//if axis is between first blade cutting upper and homing position
				IF iFb_SlaveAx.PowerOn AND iFb_SlaveAx.Position < FIRST_CUT_LOWER AND iFb_SlaveAx.Position > HOME_POS   THEN

					iBasicParSlave.Home.Mode:=4;
					iBasicParSlave.Direction:=mpAXIS_DIR_NEGATIVE ;
					iBasicParSlave.Home.HomingDirection:=mpAXIS_HOME_DIR_NEGATIVE;
					iBasicParSlave.Home.StartDirection:=1;
					iBasicParSlave.Home.SensorOffset := HOFFSET_NEGDUAL;
					iBasicParSlave.Home.HomingVelocity := HOMING_VEL;
					iBasicParSlave.Home.StartVelocity := START_VEL;
					iFb_SlaveAx.Update:=TRUE;
					iAxStep_enum := enNEGHOMING;

					//if axis is between first blade cutting upper and homing position
				ELSIF iFb_SlaveAx.PowerOn AND iFb_SlaveAx.Position < HOME_POS AND iFb_SlaveAx.Position> SEC_CUT_UPPER THEN

					iBasicParSlave.Home.Mode:=4;
					iBasicParSlave.Direction:=mpAXIS_DIR_POSITIVE ;
					iBasicParSlave.Home.HomingDirection:=mpAXIS_HOME_DIR_POSITIVE;
					iBasicParSlave.Home.StartDirection:=1;
					iBasicParSlave.Home.SensorOffset := HOFFSET_NEGDUAL;
					iBasicParSlave.Home.HomingVelocity := HOMING_VEL;
					iBasicParSlave.Home.StartVelocity := START_VEL;
					iFb_SlaveAx.Update:=TRUE;
					iAxStep_enum := enNEGHOMING;

					//if axis is between first blade cutting upper and homing position
				ELSIF iFb_SlaveAx.PowerOn AND iFb_SlaveAx.Position > FIRST_CUT_UPPER AND iFb_SlaveAx.Position < MAX_POS_AXIS THEN

					iBasicParSlave.Home.Mode:=mpAXIS_HOME_MODE_REF_PULSE;
					iBasicParSlave.Home.HomingDirection:=mpAXIS_HOME_DIR_POSITIVE;
					iBasicParSlave.Home.SensorOffset := HOFFSET_DUAL;
					iBasicParSlave.Home.HomingVelocity := 150;
					iBasicParSlave.Home.StartVelocity := 50;
					iFb_SlaveAx.Update:=TRUE;
					IF iFb_SlaveAx.UpdateDone=TRUE THEN
						iFb_SlaveAx.Home := TRUE;
						iAxStep_enum := enPOSHOMING;
						iFb_SlaveAx.Update:=FALSE;
					END_IF;
				ELSIF iFb_SlaveAx.PowerOn AND iFb_SlaveAx.Position < SEC_CUT_LOWER AND iFb_SlaveAx.Position> HOME_OFFSET THEN
					iFb_SlaveAx.Update:=TRUE;
					IF iFb_SlaveAx.UpdateDone=TRUE THEN

						iBasicParSlave.Home.Mode:=mpAXIS_HOME_MODE_REF_PULSE;
						iBasicParSlave.Home.HomingDirection:=mpAXIS_HOME_DIR_NEGATIVE;
						iBasicParSlave.Home.SensorOffset := HOFFSET_DUAL;
						iBasicParSlave.Home.HomingVelocity := HOMING_VEL;
						iBasicParSlave.Home.StartVelocity := START_VEL;
						iFb_SlaveAx.Update:=TRUE;
						IF iFb_SlaveAx.UpdateDone=TRUE THEN
							iFb_SlaveAx.Home := TRUE;
							iAxStep_enum := enPOSHOMINGSEC;
							iFb_SlaveAx.Update:=FALSE;
						END_IF;
					END_IF;
				END_IF
			END_IF

			//homing the motor
		enNEGHOMING:
			IF iFb_SlaveAx.UpdateDone=TRUE THEN
				iFb_SlaveAx.MoveAbsolute:=TRUE;
				iFb_SlaveAx.Update:=FALSE;
				iAxStep_enum :=	enNEEGHOMEMOVE;
			END_IF;

		enNEEGHOMEMOVE:
			IF iFb_SlaveAx.InPosition=TRUE THEN
				iFb_SlaveAx.MoveAbsolute:=FALSE;
				iFb_SlaveAx.Home:=TRUE;
				iAxStep_enum := enOPERATIONA;
			END_IF;

		enPOSHOMING:
			IF iFb_AxisSlave.IsHomed=TRUE THEN
				iAxStep_enum := enOPERATIONA;
			END_IF;
			//operation mode
		enPOSHOMINGSEC:

			IF iFb_AxisSlave.IsHomed=TRUE THEN
				iAxStep_enum := enOPERATIONA;
			END_IF;
			//operation mode
		enOPERATIONA:

			IF iFb_AxisSlave.IsHomed=TRUE THEN
				iFb_SlaveAx.Home:=FALSE;
			END_IF;
			//error mode
		enERRORA:
			iFb_AxisSlave.Power := FALSE;
			iFb_AxisSlave.MoveVelocity:= FALSE;
			IF iFb_SlaveAx.Error = FALSE THEN;
				iAxStep_enum := enSTARTA;
				iFb_SlaveAx.ErrorReset := FALSE;
			END_IF
	END_CASE

END_ACTION
```

#### CamAutoSingle.st - cam auto for single cutter
```iecst
(*|ŻŻŻŻŻŻŻŻŻŻŻŻŻŻŻŻŻŻŻŻŻŻŻŻŻŻŻŻŻŻŻŻŻŻŻŻŻŻŻŻŻŻŻŻŻŻŻŻŻŻŻŻŻŻŻŻŻŻŻŻŻŻŻŻŻŻŻŻŻŻŻŻŻŻŻŻŻŻŻŻŻŻŻŻŻŻŻŻŻŻŻŻŻŻŻŻŻŻŻŻŻŻŻŻŻŻŻŻŻŻ|*)
(*| Copyright      :-  B&R Industrial Automation GmbH															 |*)
(*| Contact Person :-  maskeu																					 |*)
(*|——————————————————————————————————————————————————————————————————————————————————————————————————————————————|*)
(*| System       :-  TODO: Printmark                                                                             |*)
(*| Task Name    :-  TODO: CAMAuto                                                                   	         |*)
(*| Auther Name  :-  maskeu																						 |*)
(*| Created Date :-  October 10, 2023 																		   	 |*)
(*| Task Class   :-  Task Class# Task Class No                                                                   |*)
(*| Task Time    :-  Task Timing mSec                                                                            |*)
(*| OS Version   :-  V G.9.43                                                                                    |*)
(*| AS Version   :-  AS 4.12.4.107 SPXY                                                                          |*)
(*|——————————————————————————————————————————————————————————————————————————————————————————————————————————————|*)
(*| Description  :-  TODO: Description about task                                                                |*)
(*|                                                                                                              |*)
(*|——————————————————————————————————————————————————————————————————————————————————————————————————————————————|*)
(*| History (Task Modification):                                                                                 |*)
(*|                                                                                                              |*)
(*| Version      Date       Modified By      Modification                                          Status     	 |*)
(*| V1.00.0   21/12/2023	 Maskeu        written all cam auto			                      	   Complete		 |*)
(*|______________________________________________________________________________________________________________|*)
ACTION CamSingle:
	iAx_CamSequence.Configuration.Master := ADR(gAxMaster); // Not Mplink Axis Address
	iAx_CamSequence.Configuration.MasterParID := ACP10PAR_PCTRL_S_ACT; //412 parid -

	(** STATE 0 - Event 1 - WAIT FOR TRIGGER **)

	iAx_CamSequence.Configuration.State[0].Event[0].Type :=ncTRIGGER1; //Trigger
	iAx_CamSequence.Configuration.State[0].Event[0].Attribute := ncAT_ONCE; //Reaction
	iAx_CamSequence.Configuration.State[0].Event[0].NextState := 4; //Next State

	(** STATE 4 - Event 4 - for first print mark**)
	iAx_CamSequence.Configuration.State[4].CamProfileIndex := 16#FFFE;
	iAx_CamSequence.Configuration.State[4].MasterFactor := 300 ; //Master Dist.
	iAx_CamSequence.Configuration.State[4].SlaveFactor := -400; //Slave Dist.

	iAx_CamSequence.Configuration.State[4].CompMode := ncONLYCOMP;
	iAx_CamSequence.Configuration.State[4].MasterCompDistance := 900; //Master Dist.
	iAx_CamSequence.Configuration.State[4].SlaveCompDistance :=  -1500; //Slave Dist.

	iAx_CamSequence.Configuration.State[4].Event[0].Type := ncST_END; //Trigger
	iAx_CamSequence.Configuration.State[4].Event[0].Attribute := ncST_END; //Reaction
	iAx_CamSequence.Configuration.State[4].Event[0].NextState := 5; //Next State

	(** STATE 5 - Event 5 - for first printmark linear motion**)
	iAx_CamSequence.Configuration.State[5].CamProfileIndex := 16#FFFF;
	iAx_CamSequence.Configuration.State[5].MasterFactor := 300 ; //Master Dist.
	iAx_CamSequence.Configuration.State[5].SlaveFactor := -400; //Slave Dist.

	iAx_CamSequence.Configuration.State[5].Event[0].Type := ncST_END; //Trigger
	iAx_CamSequence.Configuration.State[5].Event[0].Attribute := ncST_END; //Reaction
	iAx_CamSequence.Configuration.State[5].Event[0].NextState := 6; //Next State

	(** STATE 6 - Event 6 - for next cutting non linear motion**)
	iAx_CamSequence.Configuration.State[6].CamProfileIndex := 16#FFFE;
	iAx_CamSequence.Configuration.State[6].MasterFactor := 300 ; //Master Dist.
	iAx_CamSequence.Configuration.State[6].SlaveFactor := -400; //Slave Dist.

	iAx_CamSequence.Configuration.State[6].CompMode := ncONLYCOMP;
	iAx_CamSequence.Configuration.State[6].MasterCompDistance := 400; //Master Dist.
	iAx_CamSequence.Configuration.State[6].SlaveCompDistance :=  -3200; //Slave Dist.

	iAx_CamSequence.Configuration.State[6].Event[0].Type := ncST_END; //Trigger
	iAx_CamSequence.Configuration.State[6].Event[0].Attribute := ncST_END; //Reaction
	iAx_CamSequence.Configuration.State[6].Event[0].NextState := 2; //Next State

	(** STATE 2 - Event 2 - linear motion cutting zone**)
	iAx_CamSequence.Configuration.State[2].CamProfileIndex := 16#FFFF;
	iAx_CamSequence.Configuration.State[2].MasterFactor := 300 ; //Master Dist.
	iAx_CamSequence.Configuration.State[2].SlaveFactor := -400; //Slave Dist.

	iAx_CamSequence.Configuration.State[2].Event[0].Type := ncST_END; //Trigger
	iAx_CamSequence.Configuration.State[2].Event[0].Attribute := ncST_END; //Reaction
	iAx_CamSequence.Configuration.State[2].Event[0].NextState := 1; //Next State

	(** STATE 1 - Event 1 - non linear motion  non-cutting zone **)
	iAx_CamSequence.Configuration.State[1].CamProfileIndex := 16#FFFE;
	iAx_CamSequence.Configuration.State[1].MasterFactor := 400 ; //Master Dist.
	iAx_CamSequence.Configuration.State[1].SlaveFactor := -900; //Slave Dist.

	iAx_CamSequence.Configuration.State[1].CompMode := ncONLYCOMP;
	iAx_CamSequence.Configuration.State[1].MasterCompDistance := 400; //Master Dist.
	iAx_CamSequence.Configuration.State[1].SlaveCompDistance :=  -3200; //Slave Dist.

	iAx_CamSequence.Configuration.State[1].Event[0].Type := ncST_END; //Trigger
	iAx_CamSequence.Configuration.State[1].Event[0].Attribute := ncST_END; //Reaction
	iAx_CamSequence.Configuration.State[1].Event[0].NextState := 2; //Next State

END_ACTION
```

#### CamAutoMulti.st - cam auto for dual cutter
```iecst
(*|ŻŻŻŻŻŻŻŻŻŻŻŻŻŻŻŻŻŻŻŻŻŻŻŻŻŻŻŻŻŻŻŻŻŻŻŻŻŻŻŻŻŻŻŻŻŻŻŻŻŻŻŻŻŻŻŻŻŻŻŻŻŻŻŻŻŻŻŻŻŻŻŻŻŻŻŻŻŻŻŻŻŻŻŻŻŻŻŻŻŻŻŻŻŻŻŻŻŻŻŻŻŻŻŻŻŻŻŻŻŻ|*)
(*| Copyright      :-  B&R Industrial Automation GmbH															 |*)
(*| Contact Person :-  maskeu																					 |*)
(*|——————————————————————————————————————————————————————————————————————————————————————————————————————————————|*)
(*| System       :-  TODO: Printmark                                                                             |*)
(*| Task Name    :-  TODO: CAMAuto                                                                   	         |*)
(*| Auther Name  :-  maskeu																						 |*)
(*| Created Date :-  October 10, 2023 																		   	 |*)
(*| Task Class   :-  Task Class# Task Class No                                                                   |*)
(*| Task Time    :-  Task Timing mSec                                                                            |*)
(*| OS Version   :-  V G.9.43                                                                                    |*)
(*| AS Version   :-  AS 4.12.4.107 SPXY                                                                          |*)
(*|——————————————————————————————————————————————————————————————————————————————————————————————————————————————|*)
(*| Description  :-	 cam auto for multi or dual cutter                                                           |*)
(*|                                                                                                              |*)
(*|——————————————————————————————————————————————————————————————————————————————————————————————————————————————|*)
(*| History (Task Modification):                                                                                 |*)
(*|                                                                                                              |*)
(*| Version      Date       Modified By      Modification                                          Status     	 |*)
(*| V1.00.0   22/12/2023	 Maskeu        written all cam auto			                      	   Complete		 |*)
(*|______________________________________________________________________________________________________________|*)
ACTION CamMulti:
	iAx_CamSequence.Configuration.Master := ADR(gAxMaster); // refrencing axis
	iAx_CamSequence.Configuration.MasterParID := ACP10PAR_PCTRL_S_ACT; //412 parid -
	(** STATE 0 - Event 1 - WAIT FOR TRIGGER **)

	iAx_CamSequence.Configuration.State[0].Event[0].Type :=ncTRIGGER1 ; //Trigger
	iAx_CamSequence.Configuration.State[0].Event[0].Attribute := ncAT_ONCE; //Reaction
	iAx_CamSequence.Configuration.State[0].Event[0].NextState := 4; //Next State

	(** STATE 4 - Event 4 - first print mark non linear non cutting zone **)
	iAx_CamSequence.Configuration.State[4].CamProfileIndex := 16#FFFE;
	iAx_CamSequence.Configuration.State[4].MasterFactor := 300 ; //Master Dist.
	iAx_CamSequence.Configuration.State[4].SlaveFactor := -400; //Slave Dist.

	iAx_CamSequence.Configuration.State[4].CompMode := ncONLYCOMP;
	iAx_CamSequence.Configuration.State[4].MasterCompDistance := 900; //Master Dist.
	iAx_CamSequence.Configuration.State[4].SlaveCompDistance :=  -600; //Slave Dist.

	iAx_CamSequence.Configuration.State[4].Event[0].Type := ncST_END; //Trigger
	iAx_CamSequence.Configuration.State[4].Event[0].Attribute := ncST_END; //Reaction
	iAx_CamSequence.Configuration.State[4].Event[0].NextState := 5; //Next State

	(** STATE 5 - Event 5 - linear motion cutting zone	 **)
	iAx_CamSequence.Configuration.State[5].CamProfileIndex := 16#FFFF;
	iAx_CamSequence.Configuration.State[5].MasterFactor := 300 ; //Master Dist.
	iAx_CamSequence.Configuration.State[5].SlaveFactor := -400; //Slave Dist.

	iAx_CamSequence.Configuration.State[5].Event[0].Type := ncST_END; //Trigger
	iAx_CamSequence.Configuration.State[5].Event[0].Attribute := ncST_END; //Reaction
	iAx_CamSequence.Configuration.State[5].Event[0].NextState := 6; //Next State

	(** STATE 6 - Event 6 - non linear motion no cutting zone **)
	iAx_CamSequence.Configuration.State[6].CamProfileIndex := 16#FFFE;
	iAx_CamSequence.Configuration.State[6].MasterFactor := 300 ; //Master Dist.
	iAx_CamSequence.Configuration.State[6].SlaveFactor := -400; //Slave Dist.

	iAx_CamSequence.Configuration.State[6].CompMode := ncONLYCOMP;
	iAx_CamSequence.Configuration.State[6].MasterCompDistance := 300; //Master Dist.
	iAx_CamSequence.Configuration.State[6].SlaveCompDistance :=  -1310; //Slave Dist.

	iAx_CamSequence.Configuration.State[6].Event[0].Type := ncST_END; //Trigger
	iAx_CamSequence.Configuration.State[6].Event[0].Attribute := ncST_END; //Reaction
	iAx_CamSequence.Configuration.State[6].Event[0].NextState := 2; //Next State

	(** STATE 2 - Event 2 - linear movement in which cutting will took place **)
	iAx_CamSequence.Configuration.State[2].CamProfileIndex := 16#FFFF;
	iAx_CamSequence.Configuration.State[2].MasterFactor := 300 ; //Master Dist.
	iAx_CamSequence.Configuration.State[2].SlaveFactor := -400; //Slave Dist.

	iAx_CamSequence.Configuration.State[2].Event[0].Type := ncST_END; //Trigger
	iAx_CamSequence.Configuration.State[2].Event[0].Attribute := ncST_END; //Reaction
	iAx_CamSequence.Configuration.State[2].Event[0].NextState := 1; //Next State

	(** STATE 1 - Event 1 - non-linear movement in which cutter coming for ready to cut position **)

	iAx_CamSequence.Configuration.State[1].CamProfileIndex := 16#FFFE;
	iAx_CamSequence.Configuration.State[1].MasterFactor := 300 ; //Master Dist.
	iAx_CamSequence.Configuration.State[1].SlaveFactor := -400; //Slave Dist.

	iAx_CamSequence.Configuration.State[1].CompMode := ncONLYCOMP;
	iAx_CamSequence.Configuration.State[1].MasterCompDistance := 400; //Master Dist.
	iAx_CamSequence.Configuration.State[1].SlaveCompDistance :=  -1400; //Slave Dist.

	iAx_CamSequence.Configuration.State[1].Event[0].Type := ncST_END; //Trigger
	iAx_CamSequence.Configuration.State[1].Event[0].Attribute := ncST_END; //Reaction
	iAx_CamSequence.Configuration.State[1].Event[0].NextState := 2; //Next State

	END_ACTION
```

#### RegCap.st - reg capture 
```iecst
ACTION RegCap:

	// assinging configuration for reg capture
	iFb_RegCap.Axis					:=ADR(gAxSlave);
	iFb_RegCap.Master				:=ADR(gAxMaster);
	iFb_RegCap.AdvancedParameters 	:= iRegCapAdvPar;
	iFb_RegCap.InitData				:=TRUE;
	iFb_RegCap.SearchRM				:=TRUE;
	iFb_RegCap.Configuration		:=iRegCapConfig;
	iFb_RegCap.CutPosition			:=REAL_TO_DINT(iRegCapConfig.ProductLength);
	iFb_RegCap.Enable				:=iFb_CamSequ.InSync;
	IF iFb_AxisSlave.Info.PLCopenState= mpAXIS_SYNCHRONIZED_MOTION THEN
		iFb_RegCap();
	END_IF;
END_ACTION
```

### Program Logical/AutoCtrl/AutoCtrl (IEC)

#### Main.st - Init, cyclic, exit code
```iecst
(*|ŻŻŻŻŻŻŻŻŻŻŻŻŻŻŻŻŻŻŻŻŻŻŻŻŻŻŻŻŻŻŻŻŻŻŻŻŻŻŻŻŻŻŻŻŻŻŻŻŻŻŻŻŻŻŻŻŻŻŻŻŻŻŻŻŻŻŻŻŻŻŻŻŻŻŻŻŻŻŻŻŻŻŻŻŻŻŻŻŻŻŻŻŻŻŻŻŻŻŻŻŻŻŻŻŻŻŻŻŻŻ|*)
(*| Copyright      :-  B&R Industrial Automation GmbH															 |*)
(*| Contact Person :-  maskeu																					 |*)
(*|——————————————————————————————————————————————————————————————————————————————————————————————————————————————|*)
(*| System       :-  auto control                                                                    	 		 |*)
(*| Task Name    :-  auto control																		  		 |*)
(*| Auther Name  :-  maskeu																						 |*)
(*| Created Date :-  December 19, 2023 																		   	 |*)
(*| Task Class   :-  Task Class# 1                                                                 				 |*)
(*| Task Time    :-  Task Timing 2mSec                                                                           |*)
(*| OS Version   :-  G4.93                                                                                       |*)
(*| AS Version   :-  AS 4.12.4.107 SP                                                                            |*)
(*|——————————————————————————————————————————————————————————————————————————————————————————————————————————————|*)
(*| Description  :-  auto control- all fucniton for main control											     |*)
(*| V1.00.0   19/12/2023	 Maskeu        added pointers with homing state						Complete		 |*)
(*| V2.00.0   20/12/2023	 Maskeu        added automatic state							    Complete		 |*)
(*| V3.00.0   21/12/2023	 Maskeu        added manual state									Complete		 |*)
(*| V4.00.0   23/12/2023	 Maskeu        added cutting zone state								Complete	     |*)

PROGRAM _INIT
	//Accessing Various Variables for Pointer references
	iStatus_CutCtrl 	:= PV_xgetadr(ADR('Cutter:iCutCtrl'),ADR(CutterAdd),ADR(SizeCutter));
	iStatus_ConvCtrl 	:= PV_xgetadr(ADR('ConvCtrl:iConCtrl'),ADR(ConvAdd),ADR(SizeConv));
	iStatus_CamSeq 		:= PV_xgetadr(ADR('Cutter:iFb_CamSequ'),ADR(CamAdd),ADR(SizeCam));
	iStatus_RegCapt 	:= PV_xgetadr(ADR('Cutter:iFb_RegCap'),ADR(RegAdd),ADR(RegSize));
	iStatus_SlaveAx 	:= PV_xgetadr(ADR('Cutter:iFb_SlaveAx'),ADR(SlaveAx),ADR(SlaveSize));
	iStatus_MasterAx 	:= PV_xgetadr(ADR('ConvCtrl:iFb_MasterAx'),ADR(MasterAx),ADR(MasterSize));

END_PROGRAM

PROGRAM _CYCLIC
	(* Insert code here *)

	//Pointers Access
	pCutterCtrl		ACCESS CutterAdd;
	pConvCtrl 		ACCESS ConvAdd;
	pAx_CamSeq 		ACCESS CamAdd;
	pRegCapture 	ACCESS RegAdd;
	pMasterAx		ACCESS MasterAx;
	pSlaveAx		ACCESS SlaveAx;
	CASE iAutoCtrlState OF

		enWAIT:
			iMi_StatusTxt							:= "Please select single or dual cutter";
			pMasterAx.Enable						:=TRUE;
			pSlaveAx.Enable							:=TRUE;
			IF iAutoCtrl.Cmd.SingleCutter			=TRUE THEN
				pCutterCtrl.Cmd.SingleCutter		:=TRUE;
			ELSE
				pCutterCtrl.Cmd.SingleCutter		:=FALSE;
			END_IF;
			IF iMi_CutModeSelected=TRUE THEN
				iMi_StatusTxt						:= "Please select mode and start machine";
			END_IF;

			IF iAutoCtrl.Cmd.Start = TRUE AND iMi_CutModeSelected=TRUE THEN
				pConvCtrl.Cmd.Start 				:= TRUE;
				pCutterCtrl.Cmd.Start 				:= TRUE;
				iAutoCtrlState:=enMODE;
			END_IF;

		enMODE:
			IF gMi_ModeConfirm = TRUE THEN
				IF iAutoCtrl.Cmd.AutoMode= TRUE THEN
					iMi_SelectedMode:="Automatice Mode selected";
					iAutoCtrlState					:=enHOMING;
				ELSE
					iMi_SelectedMode:="Manual Mode Selected";
					iAutoCtrlState					:=enMANUAL;
				END_IF;
			END_IF;

			//homing for both the axis
		enHOMING:
			iMi_StatusTxt:="Homing the axis wait...";
			pAx_CamSeq.ErrorReset					:=TRUE;
			IF pMasterAx.IsHomed AND pSlaveAx.IsHomed THEN
				pAx_CamSeq.ErrorReset				:=FALSE;
				iAutoCtrlState						:=enAUTO;
			END_IF

			//autoamtic mode
		enAUTO:
			IF pAx_CamSeq.Info.MasterReady=TRUE AND  pAx_CamSeq.Info.SlaveReady=TRUE AND pAx_CamSeq.StatusID=0 THEN
				pAx_CamSeq.StartSequence			:=TRUE;
			END_IF;

			IF pAx_CamSeq.StatusID<>0 THEN
				pAx_CamSeq.ErrorReset				:=TRUE;
			ELSE
				pAx_CamSeq.ErrorReset				:=FALSE;
			END_IF;

			IF pAx_CamSeq.InSync = TRUE AND iAutoCtrl.Cmd.Start=TRUE THEN
				iMi_StatusTxt						:= " In Run Mode - Auto Mode";
				pMasterAx.MoveVelocity 				:= TRUE;
			END_IF;

			//IF stop Pressed
			IF iAutoCtrl.Cmd.Stop THEN
				iMi_StatusTxt 						:= "Stop Pressed. Press Start and select mode.";
				pMasterAx.MoveVelocity 				:= FALSE;
			END_IF

			//Disabled Cutter Cmd given
			IF iAutoCtrl.Cmd.DisableCutter=TRUE THEN
				iMi_StatusTxt := "Cutter Disabled is Pressed";
				pAx_CamSeq.StartSequence 			:= FALSE;
				pCutterCtrl.Cmd.Start 				:= FALSE;
				pSlaveAx.Power		 			:= FALSE;
				pSlaveAx.Enable 					:= FALSE;
				iAutoCtrlState			 			:= enCUT_DISABLED;
			END_IF

			//Stopping the mode and resetting machine
			IF iAutoCtrl.Cmd.ChangeMode				=TRUE AND iAutoCtrl.Cmd.Stop=TRUE THEN
				iMi_StatusTxt 						:= "Machine has Stopped";
				pMasterAx.MoveVelocity 				:= FALSE;
				iAutoCtrl.Cmd.ChangeMode			:= FALSE;
				pAx_CamSeq.StartSequence			:= FALSE;
				iAutoCtrlState 						:= enSTOP;
			END_IF

		enCUT_DISABLED:
			pCutterCtrl.Cmd.Start					:=TRUE;
			IF pSlaveAx.IsHomed=TRUE THEN
				iMi_StatusTxt:="Disabled Cutter . Restart to start";
				pSlaveAx.Home						:=FALSE;
			END_IF;

			//Stop command is Given
			IF iAutoCtrl.Cmd.Stop THEN
				pMasterAx.MoveVelocity 				:= FALSE;
			END_IF

			//Start command is given
			IF iAutoCtrl.Cmd.Start THEN
				pMasterAx.MoveVelocity				:= TRUE;
			END_IF

			//Cutter  is Enabled
			IF iAutoCtrl.Cmd.DisableCutter 			= FALSE THEN
				iMi_StatusTxt 						:= "Cutter Enabled";
				iAutoCtrlState 						:= enAUTO;
			END_IF

			//Mode has been Changed
			IF iAutoCtrl.Cmd.ChangeMode AND iAutoCtrl.Cmd.Stop THEN
				iMi_StatusTxt						:= "Machine has been Stopped";
				pMasterAx.MoveVelocity				:= FALSE;
				iAutoCtrl.Cmd.ChangeMode 			:= FALSE;
				pAx_CamSeq.StartSequence 		:= FALSE;
				iAutoCtrlState 						:= enSTOP;
			END_IF

			//Manual Mode
		enMANUAL:
			iMi_StatusTxt							:= "Manual Mode is ON";
			IF iAutoCtrl.Cmd.Stop=TRUE AND iAutoCtrl.Cmd.ChangeMode THEN
				iMi_StatusTxt						:="Machine stopped";
				iAutoCtrl.ManualCmd.ConvPowerON		:=FALSE;
				iAutoCtrl.ManualCmd.CutterPowerON	:=FALSE;
				iAutoCtrlState 						:= enSTOP;
			END_IF;

			//stopping all the fucniton
		enSTOP:
			iMi_StatusTxt							:="Machine has been stopped";
			iAutoCtrl.Cmd.Start						:=FALSE;
			gMi_ModeConfirm							:=FALSE;
			pMasterAx.Power							:=FALSE;
			pMasterAx.Enable						:=FALSE;
			pSlaveAx.Power							:=FALSE;
			pSlaveAx.Enable							:=FALSE;
			pConvCtrl.Cmd.Start						:=FALSE;
			iAutoCtrl.Cmd.ChangeMode				:=FALSE;
			iMi_CutModeSelected						:=FALSE;
			pCutterCtrl.Cmd.Start					:=FALSE;
			iAutoCtrl.Cmd.DisableCutter 			:= FALSE;
			iAutoCtrl.Cmd.Stop 						:= FALSE;
			iAutoCtrlState 							:= enWAIT;

		enCUT_ZONE:
			iMi_StatusTxt							:="Cutting Zone";
			iAutoCtrl.ManualCmd.ConvPowerON			:=FALSE;
			iAutoCtrl.ManualCmd.CutterPowerON		:=FALSE;

			IF pSlaveAx.Position > UPPER_CUT_POS OR pSlaveAx.Position < LOWER_CUT_POS THEN
				iAutoCtrl.Cmd.Start					:=FALSE;
				iAutoCtrlState						:=enWAIT;
			END_IF;

	END_CASE

	IF NOT iAutoCtrl.Cmd.AutoMode= TRUE THEN
		pMasterAx.Power								:=iAutoCtrl.ManualCmd.ConvPowerON;
		pSlaveAx.Power								:=iAutoCtrl.ManualCmd.CutterPowerON;
		pSlaveAx.JogNegative						:= pCutterCtrl.Cmd.JogBack;
		pSlaveAx.JogPositive						:=pCutterCtrl.Cmd.JogFwd;
		pMasterAx.JogPositive						:=pConvCtrl.Cmd.JogFwd;
		pMasterAx.JogNegative						:=pConvCtrl.Cmd.JogBack;
	END_IF;

	//Mapping some variables for sub task control
	pConvCtrl.Cmd.AutoMode := iAutoCtrl.Cmd.AutoMode;
	pCutterCtrl.Cmd.AutoMode := iAutoCtrl.Cmd.AutoMode;

	//Cutting zone Logic
	IF pSlaveAx.Position < UPPER_CUT_POS AND pSlaveAx.Position > LOWER_CUT_POS AND NOT iAutoCtrl.Cmd.AutoMode THEN
		iAutoCtrlState := enCUT_ZONE;
	END_IF

	//Hmi Variables calculation
	iMI_LastBagLen := pRegCapture.AdditionalInfo.ActLength / TEN;
	iMI_AvgBagLen := pRegCapture.AdditionalInfo.AverageProductLength /TEN;

	IF iAutoCtrl.Cmd.AutoMode THEN
		iMi_SelectedMode := "Auto Mode is Selected";
	ELSE
		iMi_SelectedMode := "Manual Mode is Selected";
	END_IF

	//Reset Condition
	IF iAutoCtrl.Cmd.Reset THEN
		Reset;
	END_IF

	//Condition For Calling RegMarkCapture FB
	IF pSlaveAx.Info.PLCopenState = mpAXIS_SYNCHRONIZED_MOTION THEN
		pRegCapture();
	END_IF

	//Calling Alarm ACtion file
	gMI_MODE := iAutoCtrl.Cmd.AutoMode;
	Alarms;
END_PROGRAM

END_PROGRAM

PROGRAM _EXIT
	(* Insert code here *)

END_PROGRAM
```

#### Types.typ - Local data types
```iecst
TYPE
	Reset_enum :
		( (*restting value enumaration*)
		enRESETONE, (*resting first block*)
		enRESETTWO, (*resting second block*)
		enEXIT (*exiting state*)
		);
	AutoCmd_typ : 	STRUCT  (*Auto Ctrl Command Type*)
		Start : BOOL; (*Start cmd*)
		Stop : BOOL; (*Stop cmd*)
		AutoMode : BOOL; (*Auto Mode cmd*)
		ChangeMode : BOOL; (*Change Mode cmd*)
		DisableCutter : BOOL; (*Disable Cutter cmd*)
		SingleCutter : BOOL; (*Single or Dual Cutter bit*)
		Reset : BOOL; (*Reset Complete Machine*)
	END_STRUCT;
	AutoPara_typ : 	STRUCT  (*Auto Ctrl Para Type*)
		ConvSpeed : REAL; (*Conv speed Para*)
		ConvJogSpeed : REAL; (*Conv Jog SPeed*)
		CutterJogSpeed : REAL; (*Cutter Jog Speed*)
	END_STRUCT;
	AutoManCmd_typ : 	STRUCT  (*Auto Ctrl Manaual Cmd Type*)
		ConvPowerON : BOOL; (*Conv power on*)
		CutterPowerON : BOOL; (*Cutter Power On*)
	END_STRUCT;
	AutoCtrl_typ : 	STRUCT  (*Auto Ctrl Type*)
		Cmd : AutoCmd_typ; (*Auto Ctrl cmd type*)
		Para : AutoPara_typ; (*Auto Ctrl Para type*)
		ManualCmd : AutoManCmd_typ; (*Auto Ctrl Manual Cmd Type*)
	END_STRUCT;
	AutoCtrl_enum :
		( (*Auto Ctrl State*)
		enWAIT, (*Wait state*)
		enMODE, (*Mode Select state*)
		enHOMING, (*homing State*)
		enMANUAL, (*Manual Mode*)
		enAUTO, (*Auto mode state*)
		enSTOP, (*Stop state*)
		enMAN_JOGFWD, (*Manual jog f State*)
		enMAN_JOGBWD, (*Manual jog N State*)
		enCUT_ZONE, (*Cutting zone state*)
		enCUT_DISABLED, (*Cutter Disabled STate*)
		enCUT_DISABLE_HOME (*Cutter Homing after disable*)
		);
END_TYPE
```

#### Variables.var - Local variables
```iecst
(*referecing the strcutre for pointers*)
VAR
	pCutterCtrl : REFERENCE TO AxisCtrl_typ; (*Pointer to conv ctrl*)
	pRegCapture : REFERENCE TO MC_BR_RegMarkCapture002; (*Pointer to reg capture*)
	pConvCtrl : REFERENCE TO AxisCtrl_typ; (*Pointer to Conv Ctrl*)
	pMasterAx : REFERENCE TO MpAxisBasic; (*pointer for master axis*)
	pAx_CamSeq : REFERENCE TO MpAxisCamSequencer; (*Pointer cam seq*)
	pSlaveAx : REFERENCE TO MpAxisBasic; (*pointer for slave axis*)
END_VAR
(*for pointer using size address status varibles*)
VAR
	iStatus_CutCtrl : UINT; (*status for pointer of cutter control*)
	CutterAdd : UDINT; (*cutter additon*)
	RegAdd : UDINT; (*Address*)
	RegSize : UDINT; (*Size*)
	ConvAdd : UDINT; (*Address*)
	SizeConv : UDINT; (*Address*)
	SizeCutter : UDINT; (*size of cutter*)
	iStatus_ConvCtrl : UINT; (*status of cinveyor control pointer*)
	iStatus_CamSeq : UINT; (*status of cam sequnce *)
	iStatus_RegCapt : UINT; (*status of reg capture*)
	CamAdd : UDINT; (*cam add variable*)
	SizeCam : UDINT; (*size of cam varible*)
	iStatus_SlaveAx : UDINT; (*status for slave axis pointer*)
	iStatus_MasterAx : UINT; (*status for master axis*)
	SlaveAx : UDINT; (*slave axis address*)
	MasterSize : UDINT; (*master axis size*)
	SlaveSize : UDINT; (*slave axis size*)
	MasterAx : UDINT; (*master axis address*)
END_VAR
(*enumeration  for main control state*)
VAR
	iAutoCtrlState : AutoCtrl_enum; (*Auto control state*)
END_VAR
(*resetiing the state*)
VAR
	iResetState : Reset_enum; (*restiing value enumeration -state*)
END_VAR
(*main auto control structure*)
VAR
	iAutoCtrl : AutoCtrl_typ; (*Auto ctrl struture*)
END_VAR
(*variables for hmi*)
VAR
	iMi_CutModeSelected : BOOL; (*cutter mode selected*)
	iMi_StatusTxt : WSTRING[80]; (*text on hmi for current state*)
	iMi_SelectedMode : WSTRING[80]; (*selected mode *)
	iMI_LastBagLen : REAL; (*last bag length*)
	iMI_AvgBagLen : REAL; (*average bag length*)
END_VAR
(*constants*)
VAR CONSTANT
	TEN : REAL := 10; (*ten value*)
	LIMIT_ERROR_PRODUCT : INT := 5; (*limit for error in product*)
	UPPER_CUT_POS : REAL := 3013; (*upper cutting position for first cutter*)
	LOWER_CUT_POS : REAL := 2653; (*lower cutting position for second cutter*)
END_VAR
```

#### Alarms_Reset.st - alarms and reset action
```iecst
(*|ŻŻŻŻŻŻŻŻŻŻŻŻŻŻŻŻŻŻŻŻŻŻŻŻŻŻŻŻŻŻŻŻŻŻŻŻŻŻŻŻŻŻŻŻŻŻŻŻŻŻŻŻŻŻŻŻŻŻŻŻŻŻŻŻŻŻŻŻŻŻŻŻŻŻŻŻŻŻŻŻŻŻŻŻŻŻŻŻŻŻŻŻŻŻŻŻŻŻŻŻŻŻŻŻŻŻŻŻŻŻ|*)
(*| Copyright      :-  B&R Industrial Automation GmbH															 |*)
(*| Contact Person :-  maskeu																					 |*)
(*|——————————————————————————————————————————————————————————————————————————————————————————————————————————————|*)
(*| System       :-  auto control                                                                    	 		 |*)
(*| Task Name    :-  auto control																		  		 |*)
(*| Auther Name  :-  maskeu																						 |*)
(*| Created Date :-  December 19, 2023 																		   	 |*)
(*| Task Class   :-  Task Class# 1                                                                 				 |*)
(*| Task Time    :-  Task Timing 2mSec                                                                           |*)
(*| OS Version   :-  G4.93                                                                                       |*)
(*| AS Version   :-  AS 4.12.4.107 SP                                                                            |*)
(*|——————————————————————————————————————————————————————————————————————————————————————————————————————————————|*)
(*| Description  :-  alarmsaction file				    									 					 |*)
(*| V1.00.0   23/12/2023	 Maskeu        added alarms and reset file							Complete	     |*)

ACTION Alarms:
//	in Cutting zone alarm
	IF pSlaveAx.Position < 3013 AND pSlaveAx.Position > 2653 AND NOT iAutoCtrl.Cmd.AutoMode THEN
		MpAlarmXSet(gAlarmXCore,'InTheCuttingZone');
	ELSE
		MpAlarmXReset(gAlarmXCore,'InTheCuttingZone');
	END_IF

	//Product without pritn mark limit exceeded alarm
	IF pRegCapture.ProductsWithoutRM > LIMIT_ERROR_PRODUCT THEN
		pAx_CamSeq.StartSequence 	 := FALSE;
		pMasterAx.Power					 := FALSE;
		pSlaveAx.Power					 := FALSE;
		MpAlarmXSet(gAlarmXCore,'ErrorCutting');
		iAutoCtrlState := enSTOP;
	ELSE
		MpAlarmXReset(gAlarmXCore,'ErrorCutting');
	END_IF

END_ACTION

//resetting all the values
ACTION Reset:

	CASE iResetState OF
		enRESETONE:

			iAutoCtrl.Cmd.Start 				:= FALSE;
			iAutoCtrl.Cmd.AutoMode				:= FALSE;
			iAutoCtrl.Cmd.Stop 					:= FALSE;
			iAutoCtrl.ManualCmd.ConvPowerON		:= FALSE;
			iAutoCtrl.ManualCmd.CutterPowerON 	:= FALSE;
			pMasterAx.Power 					:= FALSE;
			gMi_ModeConfirm						:= FALSE;
			pSlaveAx.Power 						:= FALSE;
			pSlaveAx.ErrorReset 				:= TRUE;
			pMasterAx.ErrorReset 				:= TRUE;
			pConvCtrl.Cmd.Start 				:= FALSE;
			pCutterCtrl.Cmd.Start 				:= FALSE;
			pAx_CamSeq.StartSequence 		:= FALSE;
			iResetState:=enRESETTWO;
		enRESETTWO:

			pMasterAx.ErrorReset 				:= FALSE;
			pMasterAx.ErrorReset 				:= FALSE;
			iAutoCtrl.Cmd.DisableCutter 		:= FALSE;
			iAutoCtrl.Cmd.SingleCutter 			:= FALSE;
			iAutoCtrl.Cmd.AutoMode 				:= FALSE;
			iMi_CutModeSelected 				:= FALSE;
			iResetState:=enEXIT;
		enEXIT:
			gMi_ModeConfirm 					:= FALSE;
			pAx_CamSeq.ErrorReset 				:= FALSE;
			pAx_CamSeq.ErrorReset 				:= TRUE;
			pMasterAx.Enable 					:= FALSE;
			pSlaveAx.Enable 					:= FALSE;
			iResetState							:=enRESETONE;
			iAutoCtrlState 						:= enWAIT ;
	END_CASE;
END_ACTION
```

### Program Logical/ConvCtrl/ConvCtrl (IEC)

#### Main.st - Init, cyclic, exit code
```iecst
(*|ŻŻŻŻŻŻŻŻŻŻŻŻŻŻŻŻŻŻŻŻŻŻŻŻŻŻŻŻŻŻŻŻŻŻŻŻŻŻŻŻŻŻŻŻŻŻŻŻŻŻŻŻŻŻŻŻŻŻŻŻŻŻŻŻŻŻŻŻŻŻŻŻŻŻŻŻŻŻŻŻŻŻŻŻŻŻŻŻŻŻŻŻŻŻŻŻŻŻŻŻŻŻŻŻŻŻŻŻŻŻ|*)
(*| Copyright      :-  B&R Industrial Automation GmbH															 |*)
(*| Contact Person :-  maskeu																					 |*)
(*|——————————————————————————————————————————————————————————————————————————————————————————————————————————————|*)
(*| System       :- conveyor control                                                                    	 	 |*)
(*| Task Name    :- conveyor control																			 |*)
(*| Auther Name  :-  maskeu																						 |*)
(*| Created Date :-  December 13, 2023 																		   	 |*)
(*| Task Class   :-  Task Class# 1                                                                 				 |*)
(*| Task Time    :-  Task Timing 10mSec                                                                          |*)
(*| OS Version   :-  V4.12.4                                                                                     |*)
(*| AS Version   :-  AS 4.12.4 .107 SP                                                                           |*)
(*|——————————————————————————————————————————————————————————————————————————————————————————————————————————————|*)
(*| Description  :-  movement of  conveyor		    															 |*)
(*| V1.00.0   22/12/2023	 Maskeu        added homing mode 									Complete	 	 |*)
(*| V2.00.0   23/12/2023	 Maskeu        added manual mode jog pos-neg						Complete		 |*)
PROGRAM _INIT
	(* Insert code here *)
	iBasicParamMaster.Acceleration:=480000;
	iBasicParamMaster.Deceleration:=4800000;
	iBasicParamMaster.Jog.Velocity:=45;
	iBasicParamMaster.Home.Mode:= mpAXIS_HOME_MODE_ABS_SWITCH;
	iBasicParamMaster.Home.StartVelocity:=200;
	iBasicParamMaster.Home.HomingDirection:= mpAXIS_HOME_DIR_POSITIVE;
	iBasicParamMaster.Home.StartDirection:=mpAXIS_HOME_DIR_POSITIVE;
	iBasicParamMaster.Home.SwitchEdge:=mpAXIS_HOME_DIR_NEGATIVE;
END_PROGRAM

PROGRAM _CYCLIC
		//linking the motor with axis
	iFb_MasterAx.Enable := 1;
	iFb_MasterAx.MpLink := ADR(gmlMaster);
	iFb_MasterAx.Axis := ADR(gAxMaster);

	iFb_MasterAx.Parameters := ADR(iBasicParamMaster);
	iFb_MasterAx();

	//Updating the paramters set from HMI by converting them
	iBasicParamMaster.Velocity := (iMI_ConSetSpeed * PRODUCT_LENGTH)/PER_SEC;
	IF iMI_ConSetSpeed <> (iBasicParamMaster.Velocity * PER_SEC)/PRODUCT_LENGTH
		OR iMI_ConSetJogAcc <> (iBasicParamMaster.Jog.Acceleration * PER_SEC)/PRODUCT_LENGTH
		OR iMI_ConSetJogDeacc <> (iBasicParamMaster.Jog.Deceleration * PER_SEC)/PRODUCT_LENGTH
		OR iMI_ConSetJogVel <> (iBasicParamMaster.Jog.Velocity  * PER_SEC)/PRODUCT_LENGTH
		THEN
		iFb_MasterAx.Update := TRUE;
		IF iFb_MasterAx.UpdateDone THEN
			iFb_MasterAx.Update := FALSE;
		END_IF
	END_IF

	//Mapping of parameters
	iBasicParamMaster.Jog.Acceleration := (iMI_ConSetJogAcc * PRODUCT_LENGTH)/PER_SEC;
	iBasicParamMaster.Jog.Deceleration := (iMI_ConSetJogDeacc * PRODUCT_LENGTH)/PER_SEC;
	iBasicParamMaster.Jog.Velocity := (iMI_ConSetJogVel * PRODUCT_LENGTH)/PER_SEC;
	iMI_ConActSpeed := (iFb_MasterAx.Velocity * PER_SEC)/PRODUCT_LENGTH ;
	//stopping the axis command
	IF	iFb_MasterAx.Stop=TRUE THEN
		IF iFb_MasterAx.Stopped=TRUE THEN
			iFb_MasterAx.Stop:=FALSE;
		END_IF;
	END_IF;

	//if axis is in error mode
	IF iFb_MasterAx.Error=TRUE THEN
		iAxStepMaster:=enERRORA;
	END_IF;

	//state neumeration for axis
	CASE iAxStepMaster OF

		//initializtion
		enINITA:
			IF iConCtrl.Cmd.Start=TRUE THEN
				iAxStepMaster := 	enSTARTA;
			END_IF;
			//starting
		enSTARTA:
			IF iFb_MasterAx.Info.ReadyToPowerOn = TRUE THEN
				iAxStepMaster := enPOWER_ONA;
			END_IF

			//poweron the axis
		enPOWER_ONA:
			iFb_MasterAx.Power 	:= TRUE;
			IF iFb_MasterAx.PowerOn THEN

				iFb_MasterAx.Home 	:= TRUE;
				IF gAutoMode =TRUE THEN
					iAxStepMaster:=enAUTOMATIC;
				ELSIF gManulMode=TRUE THEN
					iAxStepMaster:=enMANUAL;
				END_IF;
			END_IF;
			//manual mode

		enMANUAL:
			IF iConCtrl.Cmd.JogFwd THEN
				iAxStepMaster		:=	enJOGPOSITIVE;
			END_IF;

			IF iConCtrl.Cmd.JogBack THEN
				iAxStepMaster 		:= 	enJOGNEGATIVE;
			END_IF
			iVa_OldRecPosition 		:= K_ZERO;
			IF iConCtrl.Cmd.Start = FALSE THEN
				iAxStepMaster 		:= enINITA;
				iFb_MasterAx.Power := FALSE;
			END_IF

			//Jog Positive of Conv
		enJOGPOSITIVE :

			iFb_MasterAx.JogPositive := TRUE;
			IF NOT iConCtrl.Cmd.JogFwd THEN
				iFb_MasterAx.JogPositive := FALSE;
				iAxStepMaster := enMANUAL;
			END_IF

			//Jog negative of COnv
		enJOGNEGATIVE :
			iFb_MasterAx.JogNegative := TRUE;
			IF (iFb_MasterAx.JogNegative  AND EDGENEG(iConCtrl.Cmd.PrintMark)) OR
				(EDGEPOS(iFb_MasterAx.JogNegative) AND iConCtrl.Cmd.PrintMark ) THEN
				iVa_OldRecPosition := iFb_MasterAx.Position;
			END_IF
			//Setting 3 Cm limit for jog Negative
			IF (iVa_OldRecPosition - iFb_MasterAx.Position) > (PRINT_MARK_LIMIT) AND iVa_OldRecPosition <> K_ZERO THEN
				iFb_MasterAx.JogNegative := FALSE;
				iConCtrl.Cmd.JogBack := FALSE;
				iAxStepMaster := enMANUAL;
			ELSE
				iConCtrl.Status.JogNegReady := TRUE;
			END_IF

			//error mode
		enERRORA:
			iFb_MasterAx.Power := FALSE;
			iFb_MasterAx.MoveVelocity:= FALSE;
			IF iFb_MasterAx.Error = FALSE THEN;
				iAxStepMaster := enSTARTA;
				icmdErrorReset := FALSE;
			END_IF
	END_CASE

	//trigger for conveyor for homing
	iConCtrl.Cmd.PrintMark:=gIR_Trigger;
	iVa_MasterInputs.Enable:=TRUE;
	iVa_MasterInputs.Axis:=ADR(gAxMaster);
	iVa_MasterInputs.HomeSwitch:=gIR_Trigger;
	iVa_MasterInputs();

	IF iConCtrl.Cmd.Start = FALSE THEN
		iAxStepMaster := enINITA;
	END_IF

	iBasicParamMaster.CyclicRead.TorqueMode:=mpAXIS_READ_CYCLIC;
END_PROGRAM

PROGRAM _EXIT
	//DISABLING THE funciton block
	iFb_MasterAx.Enable:=FALSE;
	iFb_MasterAx();
	iVa_MasterInputs.Enable:=FALSE;
	iVa_MasterInputs();
END_PROGRAM
```

#### Types.typ - Local data types
```iecst
TYPE
	AxStep_enum :
		( (*state for axis control*)
		enINITA, (*initialize*)
		enSTARTA, (*starting axis*)
		enPOWER_ONA, (*powering on axis*)
		enAUTOMATIC, (*automatic mode*)
		enJOGPOSITIVE, (*jog positive mode*)
		enJOGNEGATIVE, (*jog negative mode*)
		enMANUAL, (*manaual mode*)
		enHOMEA, (*homing mode*)
		enOPERATIONA, (*operation mode*)
		enERRORA (*error mode*)
		);
END_TYPE
```

#### Variables.var - Local variables
```iecst
(*variables used*)
VAR
	iVl_OldVelocity : LREAL; (*old velocity for logo  conveyor*)
	iVl_OldAccNeg : REAL; (*old accelation for axis*)
	iVl_OldAcc : REAL; (*old accelartion *)
	iVa_OldRecPosition : LREAL;
	iMi_LogoNegDir : BOOL; (*negtive direction hmi button*)
	icmdUpdate : BOOL; (*update command*)
END_VAR
VAR RETAIN
	icmdStop : BOOL; (*stopping the axis*)
END_VAR
VAR
	icmdPower : BOOL; (*powering on the axis*)
END_VAR
VAR RETAIN
	icmdMoveVelocity : BOOL; (*move velocity for axis*)
END_VAR
VAR
	icmdMoveAdditive : BOOL; (*move additive axis*)
	icmdHome : BOOL; (*hooming the axis*)
	icmdErrorReset : BOOL; (*error reseting the axis*)
END_VAR
(*All the structures*)
VAR
	iBasicParamMaster : MpAxisBasicParType; (*basic parameters for axis*)
	iParamMaster : MpAxisBasicParType; (*parameters for slave*)
	iRegCapAdvPar : ACP10APNWCPA_typ; (*reg capture advance parameters*)
	iConCtrl : AxisCtrl_typ; (*axis control structure*)
	iFb_BasicInfo : MpAxisBasicInfoType; (*basic info structure*)
	iParaSlave : MpAxisBasicParType; (*prameters for slave*)
END_VAR
(*all the function blocks*)
VAR
	iAx_CamSequence : MpAxisCamSequencerParType; (*Cam Seq Structure*)
	iFb_RegCap : MC_BR_RegMarkCapture002; (*reg capture fucntion *)
	iVa_MasterInputs : MC_BR_SetHardwareInputs; (*input from the ir sensor*)
	iRegCapConfig : MC_BR_CFG_RM2_REF; (*reg capture configuration*)
	iFb_MC_MoveVelocity_0 : MC_MoveVelocity; (*funciton bloack for velocity*)
	iFb_MasterAx : MpAxisBasic; (*basic function for axis*)
	iFb_CamSequ : MpAxisCamSequencer; (*cam sequencer fucntinon*)
END_VAR
(*enumeration for axis control*)
VAR
	iAxStepMaster : AxStep_enum; (*steps for logo conveyor*)
END_VAR
(*all constants *)
VAR CONSTANT
	HOMING_VEL : REAL := 500; (*homing velocity for axis*)
	HOFFSET_SINGLE : REAL := 1033; (*offset for axis*)
	ZEROSPD : REAL := 0; (*zero speed to assign*)
	UPPER_CUT_POS : LREAL := 3013; (*upper cutting position*)
	START_VEL : REAL := 145; (*starting velocity*)
	INIT_THOUSAND : REAL := 1000; (*inital value thousand*)
	PRODUCT_LENGTH : REAL := 700.0; (*Product length*)
	PER_SEC : REAL := 60.0; (*Per Sec*)
	INIT_FTHOUSAND : REAL := 5000; (*inital five thousand *)
	INIT_FIHNRD : REAL := 500; (*inital value five hundread*)
	SPEED : REAL := 0.25; (*speed*)
	SCALSPEEDTEN : REAL := 10000; (*scaling of speed*)
	PRINT_MARK_LIMIT : LREAL := 300; (*print mark limit*)
	LOWER_CUT_POS : LREAL := 2653; (*lower cutting position*)
	K_ZERO : LREAL := 0.0; (*zero value*)
END_VAR
VAR
	HOFFSET_DUAL : LREAL := 133; (*offset value for dual cutter*)
END_VAR
(*for hmi variables*)
VAR
	iMI_ConSetSpeed : REAL := 120; (*Conv Set Speed*)
	iMI_ConActSpeed : REAL; (*Conv act speed*)
	iMI_ConSetJogAcc : REAL := 300; (*Conv Set jog speed*)
	iMI_ConSetJogDeacc : REAL := 300; (*Conv set jog deaccleration*)
	iMI_ConSetJogVel : REAL := 60; (*Conv Set jog acceleration*)
END_VAR
```

#### ConvAxis.st
```iecst
(*|ŻŻŻŻŻŻŻŻŻŻŻŻŻŻŻŻŻŻŻŻŻŻŻŻŻŻŻŻŻŻŻŻŻŻŻŻŻŻŻŻŻŻŻŻŻŻŻŻŻŻŻŻŻŻŻŻŻŻŻŻŻŻŻŻŻŻŻŻŻŻŻŻŻŻŻŻŻŻŻŻŻŻŻŻŻŻŻŻŻŻŻŻŻŻŻŻŻŻŻŻŻŻŻŻŻŻŻŻŻŻ|*)
(*| Copyright      :-  B&R Industrial Automation GmbH															 |*)
(*| Contact Person :-  maskeu																					 |*)
(*|——————————————————————————————————————————————————————————————————————————————————————————————————————————————|*)
(*| System       :-  TODO:logo conv axis                                                                      	 |*)
(*| Task Name    :-  TODO: logo conv axis																		 |*)
(*| Auther Name  :-  maskeu																						 |*)
(*| Created Date :-  December 13, 2023 																		   	 |*)
(*| Task Class   :-  Task Class# 1                                                                 				 |*)
(*| Task Time    :-  Task Timing 10mSec                                                                          |*)
(*| OS Version   :-  V4.12.4                                                                                     |*)
(*| AS Version   :-  AS 4.12.4 .107 SP                                                                           |*)
(*|——————————————————————————————————————————————————————————————————————————————————————————————————————————————|*)
(*| Description  :-  TODO: basic movement of axis with the conveyor		    									 |*)

ACTION ConvAXisAxn:
	//linking the motor with axis
	iFb_MasterAx.Enable := 1;
	iFb_MasterAx.MpLink := ADR(gmlSlave);
	iFb_MasterAx.Axis := ADR(gAxSlave);

	iFb_MasterAx.Parameters := ADR(iBasicParameters);
	iFb_MasterAx();

	//	if new velocity by user input is different then will update
	//	IF iVl_OldVelocity <> iBasicParameters.Acceleration THEN
	//		iFb_MasterAx.Update:=TRUE ;
	//		IF	iFb_MasterAx.UpdateDone=TRUE THEN
	//			iVl_OldVelocity:= iBasicParameters.Velocity;
	//			iFb_MasterAx.Update:=FALSE ;
	//		END_IF;
	//	END_IF;
	//
	//	//	if new accelaration by user input is different then will update
	//	IF iVl_OldAcc<> iBasicParameters.Acceleration THEN
	//		iFb_MasterAx.Update:=TRUE ;
	//		IF	iFb_MasterAx.UpdateDone=TRUE THEN
	//			iVl_OldAcc:= iBasicParameters.Acceleration;
	//			iFb_MasterAx.Update:=FALSE ;
	//		END_IF;
	//	END_IF;
	//
	//	//	if new deccelaration by user input is different then will update
	//	IF iVl_OldAccNeg<> iBasicParameters.Deceleration THEN
	//		iFb_MasterAx.Update:=TRUE ;
	//		IF	iFb_MasterAx.UpdateDone=TRUE THEN
	//			iVl_OldAccNeg:= iBasicParameters.Deceleration;
	//			iFb_MasterAx.Update:=FALSE ;
	//		END_IF;
	//	END_IF;

	//Limit for the torque
	iBasicParameters.Torque.Limit:=0.8;

	//stopping the axis command
	IF icmdStop=TRUE THEN
		iFb_MasterAx.Stop:=TRUE;
		IF iFb_MasterAx.Stopped=TRUE THEN
			iFb_MasterAx.Stop:=FALSE;
			icmdStop:=FALSE;
		END_IF;
	END_IF;

	//if axis is in error mode
	IF iFb_MasterAx.Error=TRUE THEN
		iAxStep_enum:=enERRORA;
	END_IF;

	//state neumeration for axis
	CASE iAxStep_enum OF

		//initializtion
		enINITA:
			iAxStep_enum := 	enSTARTA;

			//starting
		enSTARTA:
			IF iFb_MasterAx.Info.ReadyToPowerOn = TRUE THEN
				iAxStep_enum := enPOWER_ONA;
			END_IF

			//poweron the axis
		enPOWER_ONA:
			icmdPower := TRUE;
			IF iFb_MasterAx.PowerOn = TRUE THEN
				IF iFb_MasterAx.PowerOn AND iFb_MasterAx.Position < LOWER_CUT_POS THEN
					icmdUpdate:=TRUE;
					IF iFb_MasterAx.UpdateDone=TRUE THEN
						iAxStep_enum := enNEGHOMING;
						icmdUpdate:=FALSE;
					END_IF;
				END_IF
				IF iFb_MasterAx.PowerOn AND iFb_MasterAx.Position > UPPER_CUT_POS THEN
					icmdUpdate:=TRUE;
					IF iFb_MasterAx.UpdateDone=TRUE THEN
						iAxStep_enum := enPOSHOMING;
						icmdUpdate:=FALSE;
					END_IF;
				END_IF
			END_IF

			//homing the motor
		enNEGHOMING:
			iBasicParameters.Home.Mode:=mpAXIS_HOME_MODE_REF_PULSE;
			iBasicParameters.Home.HomingDirection:=mpAXIS_HOME_DIR_NEGATIVE;
			iBasicParameters.Home.SensorOffset := HOFFSET_SINGLE;
			iBasicParameters.Home.HomingVelocity := HOMING_VEL;
			iBasicParameters.Home.StartVelocity := START_VEL;

			icmdHome := TRUE;
		enPOSHOMING:
			iBasicParameters.Home.Mode:=mpAXIS_HOME_MODE_REF_PULSE;
			iBasicParameters.Home.HomingDirection:=mpAXIS_HOME_DIR_POSITIVE;;
			iBasicParameters.Home.SensorOffset := HOFFSET_SINGLE;
			iBasicParameters.Home.HomingVelocity := HOMING_VEL;
			iBasicParameters.Home.StartVelocity := START_VEL;

			icmdHome := TRUE;
			//operation mode
		enOPERATIONA:

			IF iFb_MasterAx.IsHomed=TRUE THEN
				icmdHome := FALSE;
				iAxStep_enum:=enOPERATIONA;
			END_IF;

			IF iFb_MasterAx.Error =TRUE THEN
				iAxStep_enum := enERRORA;
			END_IF
			IF icmdMoveAdditive=TRUE THEN
				iFb_MasterAx.MoveAdditive:=TRUE;
				icmdMoveAdditive := FALSE;
				icmdHome := FALSE;
			END_IF;

			//error mode
		enERRORA:
			icmdPower := FALSE;
			icmdMoveVelocity := FALSE;
			icmdStop := FALSE;

			icmdErrorReset:=TRUE;
			IF iFb_MasterAx.Error = FALSE THEN;
				iAxStep_enum := enSTARTA;
				icmdErrorReset := FALSE;
			END_IF
	END_CASE
	iFb_MasterAx.Update:=icmdUpdate;
	iFb_MasterAx.Home:=icmdHome;
	iFb_MasterAx.Power:=icmdPower;

END_ACTION
```

### Program Logical/Alarms/AlarmsX (IEC)

#### Variables.var
```iecst
(*For HMI history of alarms*)
VAR
	iFb_AlarmHistory : MpAlarmXHistory; (*alarms histrory*)
END_VAR
(*HMI visu active and pending alarms*)
VAR
	iFb_AlarmX : MpAlarmXCore; (*alarm x core fucniton block*)
END_VAR
```

#### Main.st
```iecst
(*|ŻŻŻŻŻŻŻŻŻŻŻŻŻŻŻŻŻŻŻŻŻŻŻŻŻŻŻŻŻŻŻŻŻŻŻŻŻŻŻŻŻŻŻŻŻŻŻŻŻŻŻŻŻŻŻŻŻŻŻŻŻŻŻŻŻŻŻŻŻŻŻŻŻŻŻŻŻŻŻŻŻŻŻŻŻŻŻŻŻŻŻŻŻŻŻŻŻŻŻŻŻŻŻŻŻŻŻŻŻŻ|*)
(*| Copyright      :-  B&R Industrial Automation GmbH															 |*)
(*| Contact Person :-  maskeu																					 |*)
(*|——————————————————————————————————————————————————————————————————————————————————————————————————————————————|*)
(*| System       :-  alarms Control  	                                                                         |*)
(*| Task Name    :-  alarms Control                                                                    	         |*)
(*| Auther Name  :-  maskeu																						 |*)
(*| Created Date :-  October 10, 2023 																		   	 |*)
(*| Task Class   :-  Task Class #1                                                                               |*)
(*| Task Time    :-  Task Timing 10mSec                                                                          |*)
(*| OS Version   :-  G 4.93	                                                                                     |*)
(*| AS Version   :-  AS 4.12.4.107 SP                                                                            |*)
(*|——————————————————————————————————————————————————————————————————————————————————————————————————————————————|*)
(*| Description  :-  alarms Control                                                            					 |*)
(*|                                                                                                              |*)
(*|——————————————————————————————————————————————————————————————————————————————————————————————————————————————|*)
(*| History (Task Modification):                                                                                 |*)
(*|                                                                                                              |*)
(*| V1.00.0   23/12/2023    maskeu        added alarms fucntion block	                       compelete	     |*)

PROGRAM _INIT

	//if any errors then will be removed
	iFb_AlarmX.ErrorReset:=TRUE;
	iFb_AlarmX();
END_PROGRAM

PROGRAM _CYCLIC

	// alarmx on
	iFb_AlarmX.Enable:=TRUE;
	iFb_AlarmX.MpLink:=ADR(gAlarmXCore);
	iFb_AlarmX();

END_PROGRAM

PROGRAM _EXIT
	//Disabling the function block
	iFb_AlarmX.Enable:=FALSE;
	iFb_AlarmX();
END_PROGRAM
```

### Program Logical/Datarec/DataRec (IEC)

#### Variables.var
```iecst
VAR
	iFB_DataR : MpDataRecorder; (*Data recorder FB*)
	iFB_DataRegPar : MpDataRegPar; (*Data Recorder Reg Par FB *)
END_VAR
```

#### Main.st
```iecst
(*|ŻŻŻŻŻŻŻŻŻŻŻŻŻŻŻŻŻŻŻŻŻŻŻŻŻŻŻŻŻŻŻŻŻŻŻŻŻŻŻŻŻŻŻŻŻŻŻŻŻŻŻŻŻŻŻŻŻŻŻŻŻŻŻŻŻŻŻŻŻŻŻŻŻŻŻŻŻŻŻŻŻŻŻŻŻŻŻŻŻŻŻŻŻŻŻŻŻŻŻŻŻŻŻŻŻŻŻŻŻŻ|*)
(*| Copyright      :-  B&R Industrial Automation GmbH															 |*)
(*| Contact Person :-  maskeu																					 |*)
(*|——————————————————————————————————————————————————————————————————————————————————————————————————————————————|*)
(*| System       :-  data recorder																				 |*)
(*| Task Name    :-  data control																		  		 |*)
(*| Auther Name  :-  maskeu																						 |*)
(*| Created Date :-  December 19, 2023 																		   	 |*)
(*| Task Class   :-  Task Class# 1                                                                 				 |*)
(*| Task Time    :-  Task Timing 2mSec                                                                           |*)
(*| OS Version   :-  G4.93                                                                                       |*)
(*| AS Version   :-  AS 4.12.4.107 SP                                                                            |*)
(*|——————————————————————————————————————————————————————————————————————————————————————————————————————————————|*)
(*| Description  :-  CUTTER cam sequnce and basic initial prameters		    									 |*)
(*| V1.00.0   23/12/2023	 Maskeu        added data recorder 									Complete		 |*)

PROGRAM _INIT

END_PROGRAM

PROGRAM _CYCLIC

	//fucntion block for data recorder
	iFB_DataR.DeviceName 		:= ADR('USER');
	iFB_DataR.Enable 			:= TRUE;
	iFB_DataR.MpLink 			:= ADR(gDataRecorder);
	iFB_DataR.SamplingTime 		:= T#1s;
	iFB_DataR.Record 			:= TRUE;
	iFB_DataR.RecordMode		:= mpDATA_RECORD_MODE_VALUE;

	iFB_DataR();

	//data reg par parameters
	iFB_DataRegPar.Enable		:= TRUE;
	iFB_DataRegPar.MpLink 		:= ADR(gDataRecorder);
	iFB_DataRegPar.PVName 		:= ADR('AutoCtrl:iMI_AvgBagLen');
	iFB_DataRegPar();

END_PROGRAM

PROGRAM _EXIT
	//Diabling   fucniton block
	iFB_DataR.Enable := FALSE;
	iFB_DataRegPar.Enable := FALSE;
	iFB_DataR();
	iFB_DataRegPar();
END_PROGRAM
```

- Visualisation Logical/Visu (not shown)

- Visualisation Logical/mappView (not shown)

Listed in the project but not available here: Logical/Axis/acp10etxen, Logical/Axis/gAxSlave/gAxSlavea, Logical/Cutter/CutCtrl.typ
